LIN {X 0,Y 573.624,Z 371.5,A -85,B 0,C 180,E1 -2266.777,E2 -2266.777} C_VEL
LIN {X 0,Y 573.867,Z 351.071,A -85,B 0,C 180,E1 -2269.438,E2 -2269.438} C_VEL
LIN {X 0,Y 574.138,Z 330.864,A -85,B 0,C 180,E1 -2272.111,E2 -2272.111} C_VEL
LIN {X 0,Y 574.251,Z 318.107,A -85,B 0,C 180,E1 -2273.82,E2 -2273.82} C_VEL
LIN {X 0,Y 573.282,Z 312.704,A -85,B 0,C 180,E1 -2274.609,E2 -2274.609} C_VEL
LIN {X 0,Y 573.246,Z 312.705,A -85,B 0,C 180,E1 -2276.975,E2 -2276.975} C_VEL
LIN {X 0,Y 573.246,Z 312.7,A -85,B 0,C 180,E1 -2279.488,E2 -2279.488} C_VEL
LIN {X 0,Y 573.251,Z 312.707,A -85,B 0,C 180,E1 -2282.644,E2 -2282.644} C_VEL
LIN {X 0,Y 573.249,Z 312.699,A -85,B 0,C 180,E1 -2285.184,E2 -2285.184} C_VEL
LIN {X 0,Y 573.231,Z 312.7,A -85,B 0,C 180,E1 -2287.807,E2 -2287.807} C_VEL
LIN {X 0,Y 573.238,Z 312.706,A -85,B 0,C 180,E1 -2290.524,E2 -2290.524} C_VEL
LIN {X 0,Y 573.232,Z 312.699,A -85,B 0,C 180,E1 -2293.358,E2 -2293.358} C_VEL
LIN {X 0,Y 573.236,Z 312.708,A -85,B 0,C 180,E1 -2296.33,E2 -2296.33} C_VEL
LIN {X 0,Y 573.233,Z 312.705,A -85,B 0,C 180,E1 -2298.543,E2 -2298.543} C_VEL
LIN {X 0,Y 573.231,Z 312.701,A -85,B 0,C 180,E1 -2301.298,E2 -2301.298} C_VEL
LIN {X 0,Y 573.229,Z 312.709,A -85,B 0,C 180,E1 -2304.014,E2 -2304.014} C_VEL
LIN {X 0,Y 573.258,Z 312.7,A -85,B 0,C 180,E1 -2306.517,E2 -2306.517} C_VEL
LIN {X 0,Y 573.214,Z 312.701,A -85,B 0,C 180,E1 -2309.118,E2 -2309.118} C_VEL
LIN {X 0,Y 573.213,Z 312.703,A -85,B 0,C 180,E1 -2311.434,E2 -2311.434} C_VEL
LIN {X 0,Y 573.229,Z 312.701,A -85,B 0,C 180,E1 -2314.589,E2 -2314.589} C_VEL
LIN {X 0,Y 573.216,Z 312.709,A -85,B 0,C 180,E1 -2317.661,E2 -2317.661} C_VEL
LIN {X 0,Y 573.252,Z 312.698,A -85,B 0,C 180,E1 -2320.67,E2 -2320.67} C_VEL
LIN {X 0,Y 573.221,Z 312.71,A -85,B 0,C 180,E1 -2323.621,E2 -2323.621} C_VEL
LIN {X 0,Y 573.245,Z 312.706,A -85,B 0,C 180,E1 -2325.806,E2 -2325.806} C_VEL
LIN {X 0,Y 573.21,Z 312.702,A -85,B 0,C 180,E1 -2328.764,E2 -2328.764} C_VEL
LIN {X 0,Y 573.219,Z 312.711,A -85,B 0,C 180,E1 -2331.54,E2 -2331.54} C_VEL
LIN {X 0,Y 573.245,Z 312.699,A -85,B 0,C 180,E1 -2334.372,E2 -2334.372} C_VEL
LIN {X 0,Y 573.283,Z 312.7,A -85,B 0,C 180,E1 -2337.189,E2 -2337.189} C_VEL
LIN {X 0,Y 573.285,Z 312.695,A -85,B 0,C 180,E1 -2340,E2 -2340} C_VEL
LIN {X 0,Y 573.275,Z 312.696,A -85,B 0,C 180,E1 -2342.811,E2 -2342.811} C_VEL
LIN {X 0,Y 573.272,Z 312.699,A -85,B 0,C 180,E1 -2345.629,E2 -2345.629} C_VEL
LIN {X 0,Y 573.252,Z 312.699,A -85,B 0,C 180,E1 -2347.751,E2 -2347.751} C_VEL
LIN {X 0,Y 573.229,Z 312.703,A -85,B 0,C 180,E1 -2350.598,E2 -2350.598} C_VEL
LIN {X 0,Y 573.223,Z 312.704,A -85,B 0,C 180,E1 -2352.75,E2 -2352.75} C_VEL
LIN {X 0,Y 573.216,Z 312.71,A -85,B 0,C 180,E1 -2354.921,E2 -2354.921} C_VEL
LIN {X 0,Y 573.225,Z 312.701,A -85,B 0,C 180,E1 -2357.849,E2 -2357.849} C_VEL
LIN {X 0,Y 573.228,Z 312.7,A -85,B 0,C 180,E1 -2360.078,E2 -2360.078} C_VEL
LIN {X 0,Y 573.223,Z 312.703,A -85,B 0,C 180,E1 -2362.339,E2 -2362.339} C_VEL
LIN {X 0,Y 573.234,Z 312.702,A -85,B 0,C 180,E1 -2364.358,E2 -2364.358} C_VEL
LIN {X 0,Y 572.608,Z 312.787,A -85,B 0,C 180,E1 -2364.944,E2 -2364.944} C_VEL
LIN {X 0,Y 569.771,Z 313.141,A -85,B 0,C 180,E1 -2365.895,E2 -2365.895} C_VEL
LIN {X 0,Y 567.341,Z 313.441,A -85,B 0,C 180,E1 -2366.661,E2 -2366.661} C_VEL
LIN {X 0,Y 566.286,Z 313.569,A -85,B 0,C 180,E1 -2367.252,E2 -2367.252} C_VEL
LIN {X 0,Y 566.195,Z 313.578,A -85,B 0,C 180,E1 -2367.452,E2 -2367.452} C_VEL
LIN {X 0,Y 566.189,Z 313.578,A -85,B 0,C 180,E1 -2369.77,E2 -2369.77} C_VEL
LIN {X 0,Y 566.198,Z 313.581,A -85,B 0,C 180,E1 -2372.431,E2 -2372.431} C_VEL
LIN {X 0,Y 566.179,Z 313.583,A -85,B 0,C 180,E1 -2374.991,E2 -2374.991} C_VEL
LIN {X 0,Y 566.189,Z 313.577,A -85,B 0,C 180,E1 -2377.462,E2 -2377.462} C_VEL
LIN {X 0,Y 566.221,Z 313.578,A -85,B 0,C 180,E1 -2380.198,E2 -2380.198} C_VEL
LIN {X 0,Y 566.201,Z 313.578,A -85,B 0,C 180,E1 -2383.055,E2 -2383.055} C_VEL
LIN {X 0,Y 566.191,Z 313.582,A -85,B 0,C 180,E1 -2386.05,E2 -2386.05} C_VEL
LIN {X 0,Y 566.218,Z 313.575,A -85,B 0,C 180,E1 -2389.214,E2 -2389.214} C_VEL
LIN {X 0,Y 566.187,Z 313.58,A -85,B 0,C 180,E1 -2391.638,E2 -2391.638} C_VEL
LIN {X 0,Y 566.198,Z 313.585,A -85,B 0,C 180,E1 -2394.312,E2 -2394.312} C_VEL
LIN {X 0,Y 566.229,Z 313.575,A -85,B 0,C 180,E1 -2396.899,E2 -2396.899} C_VEL
LIN {X 0,Y 566.182,Z 313.581,A -85,B 0,C 180,E1 -2399.408,E2 -2399.408} C_VEL
LIN {X 0,Y 566.267,Z 313.716,A -85,B 0,C 180,E1 -2402.514,E2 -2402.514} C_VEL
LIN {X 0,Y 566.832,Z 317.946,A -85,B 0,C 180,E1 -2403.217,E2 -2403.217} C_VEL
LIN {X 0,Y 566.597,Z 335.971,A -85,B 0,C 180,E1 -2406.033,E2 -2406.033} C_VEL
LIN {X 0,Y 566.549,Z 342.685,A -85,B 0,C 180,E1 -2407.072,E2 -2407.072} C_VEL
LIN {X 0,Y 567.797,Z 350.391,A -85,B 0,C 180,E1 -2407.22,E2 -2407.22} C_VEL
LIN {X 0,Y 567.418,Z 479.258,A -85,B 0,C 180,E1 -2408.888,E2 -2408.888} C_VEL
LIN {X 0,Y 567.304,Z 493.234,A -85,B 0,C 180,E1 -2409.207,E2 -2409.207} C_VEL
LIN {X 0,Y 567.147,Z 507.772,A -85,B 0,C 180,E1 -2409.698,E2 -2409.698} C_VEL
LIN {X 0,Y 566.966,Z 520.604,A -85,B 0,C 180,E1 -2410.278,E2 -2410.278} C_VEL
LIN {X 0,Y 566.796,Z 533.294,A -85,B 0,C 180,E1 -2411.005,E2 -2411.005} C_VEL
LIN {X 0,Y 566.583,Z 545.097,A -85,B 0,C 180,E1 -2411.842,E2 -2411.842} C_VEL
LIN {X 0,Y 566.392,Z 556.565,A -85,B 0,C 180,E1 -2412.834,E2 -2412.834} C_VEL
LIN {X 0,Y 566.255,Z 565.673,A -85,B 0,C 180,E1 -2413.785,E2 -2413.785} C_VEL
LIN {X 0,Y 566.162,Z 574.547,A -85,B 0,C 180,E1 -2414.89,E2 -2414.89} C_VEL
LIN {X 0,Y 566.053,Z 582.989,A -85,B 0,C 180,E1 -2416.173,E2 -2416.173} C_VEL
LIN {X 0,Y 565.957,Z 589.719,A -85,B 0,C 180,E1 -2417.449,E2 -2417.449} C_VEL
LIN {X 0,Y 565.963,Z 595.363,A -85,B 0,C 180,E1 -2418.817,E2 -2418.817} C_VEL
LIN {X 0,Y 565.925,Z 599.074,A -85,B 0,C 180,E1 -2419.988,E2 -2419.988} C_VEL
LIN {X 0,Y 565.854,Z 602.252,A -85,B 0,C 180,E1 -2421.429,E2 -2421.429} C_VEL
LIN {X 0,Y 565.886,Z 604.025,A -85,B 0,C 180,E1 -2422.866,E2 -2422.866} C_VEL
LIN {X 0,Y 565.898,Z 604.451,A -85,B 0,C 180,E1 -2424.298,E2 -2424.298} C_VEL
LIN {X 0,Y 565.91,Z 603.55,A -85,B 0,C 180,E1 -2425.727,E2 -2425.727} C_VEL
LIN {X 0,Y 565.872,Z 601.307,A -85,B 0,C 180,E1 -2427.152,E2 -2427.152} C_VEL
LIN {X 0,Y 565.869,Z 597.676,A -85,B 0,C 180,E1 -2428.577,E2 -2428.577} C_VEL
LIN {X 0,Y 565.914,Z 592.561,A -85,B 0,C 180,E1 -2430,E2 -2430} C_VEL
LIN {X 0,Y 566.006,Z 587.613,A -85,B 0,C 180,E1 -2431.067,E2 -2431.067} C_VEL
LIN {X 0,Y 566.042,Z 580.556,A -85,B 0,C 180,E1 -2432.313,E2 -2432.313} C_VEL
LIN {X 0,Y 566.184,Z 573.191,A -85,B 0,C 180,E1 -2433.38,E2 -2433.38} C_VEL
LIN {X 0,Y 566.313,Z 564.376,A -85,B 0,C 180,E1 -2434.448,E2 -2434.448} C_VEL
LIN {X 0,Y 566.456,Z 553.745,A -85,B 0,C 180,E1 -2435.518,E2 -2435.518} C_VEL
LIN {X 0,Y 566.63,Z 543.012,A -85,B 0,C 180,E1 -2436.409,E2 -2436.409} C_VEL
LIN {X 0,Y 566.798,Z 530.428,A -85,B 0,C 180,E1 -2437.267,E2 -2437.267} C_VEL
LIN {X 0,Y 567.034,Z 518.388,A -85,B 0,C 180,E1 -2437.925,E2 -2437.925} C_VEL
LIN {X 0,Y 567.209,Z 504.85,A -85,B 0,C 180,E1 -2438.506,E2 -2438.506} C_VEL
LIN {X 0,Y 567.387,Z 490.587,A -85,B 0,C 180,E1 -2438.952,E2 -2438.952} C_VEL
LIN {X 0,Y 567.466,Z 476.634,A -85,B 0,C 180,E1 -2439.242,E2 -2439.242} C_VEL
LIN {X 0,Y 567.739,Z 349.084,A -85,B 0,C 180,E1 -2440.889,E2 -2440.889} C_VEL
LIN {X 0,Y 566.57,Z 342.666,A -85,B 0,C 180,E1 -2441.021,E2 -2441.021} C_VEL
LIN {X 0,Y 566.763,Z 324.714,A -85,B 0,C 180,E1 -2443.81,E2 -2443.81} C_VEL
LIN {X 0,Y 566.778,Z 316.589,A -85,B 0,C 180,E1 -2445.093,E2 -2445.093} C_VEL
LIN {X 0,Y 566.204,Z 313.585,A -85,B 0,C 180,E1 -2445.616,E2 -2445.616} C_VEL
LIN {X 0,Y 566.206,Z 313.585,A -85,B 0,C 180,E1 -2448.077,E2 -2448.077} C_VEL
LIN {X 0,Y 566.21,Z 313.58,A -85,B 0,C 180,E1 -2450.337,E2 -2450.337} C_VEL
LIN {X 0,Y 566.172,Z 313.582,A -85,B 0,C 180,E1 -2453.28,E2 -2453.28} C_VEL
LIN {X 0,Y 566.217,Z 313.584,A -85,B 0,C 180,E1 -2455.748,E2 -2455.748} C_VEL
LIN {X 0,Y 566.204,Z 313.578,A -85,B 0,C 180,E1 -2458.201,E2 -2458.201} C_VEL
LIN {X 0,Y 566.195,Z 313.579,A -85,B 0,C 180,E1 -2461.076,E2 -2461.076} C_VEL
LIN {X 0,Y 566.213,Z 313.583,A -85,B 0,C 180,E1 -2463.733,E2 -2463.733} C_VEL
LIN {X 0,Y 566.207,Z 313.575,A -85,B 0,C 180,E1 -2466.568,E2 -2466.568} C_VEL
LIN {X 0,Y 566.219,Z 313.578,A -85,B 0,C 180,E1 -2469.685,E2 -2469.685} C_VEL
LIN {X 0,Y 566.197,Z 313.578,A -85,B 0,C 180,E1 -2472.916,E2 -2472.916} C_VEL
LIN {X 0,Y 566.194,Z 313.578,A -85,B 0,C 180,E1 -2476.048,E2 -2476.048} C_VEL
LIN {X 0,Y 566.198,Z 313.583,A -85,B 0,C 180,E1 -2479.213,E2 -2479.213} C_VEL
LIN {X 0,Y 566.178,Z 313.582,A -85,B 0,C 180,E1 -2481.636,E2 -2481.636} C_VEL
LIN {X 0,Y 566.157,Z 313.582,A -85,B 0,C 180,E1 -2484.307,E2 -2484.307} C_VEL
LIN {X 0,Y 566.195,Z 313.581,A -85,B 0,C 180,E1 -2486.896,E2 -2486.896} C_VEL
LIN {X 0,Y 566.169,Z 313.586,A -85,B 0,C 180,E1 -2489.406,E2 -2489.406} C_VEL
LIN {X 0,Y 566.202,Z 313.574,A -85,B 0,C 180,E1 -2491.856,E2 -2491.856} C_VEL
LIN {X 0,Y 566.194,Z 313.576,A -85,B 0,C 180,E1 -2494.25,E2 -2494.25} C_VEL
LIN {X 0,Y 566.161,Z 313.584,A -85,B 0,C 180,E1 -2497.367,E2 -2497.367} C_VEL
LIN {X 0,Y 566.191,Z 313.575,A -85,B 0,C 180,E1 -2499.662,E2 -2499.662} C_VEL
LIN {X 0,Y 566.179,Z 313.584,A -85,B 0,C 180,E1 -2502.667,E2 -2502.667} C_VEL
LIN {X 0,Y 566.2,Z 313.575,A -85,B 0,C 180,E1 -2505.626,E2 -2505.626} C_VEL
LIN {X 0,Y 566.219,Z 313.579,A -85,B 0,C 180,E1 -2508.676,E2 -2508.676} C_VEL
LIN {X 0,Y 566.177,Z 313.58,A -85,B 0,C 180,E1 -2511.433,E2 -2511.433} C_VEL
LIN {X 0,Y 566.233,Z 313.575,A -85,B 0,C 180,E1 -2514.301,E2 -2514.301} C_VEL
LIN {X 0,Y 566.245,Z 313.57,A -85,B 0,C 180,E1 -2517.866,E2 -2517.866} C_VEL
LIN {X 0,Y 566.285,Z 313.572,A -85,B 0,C 180,E1 -2520.711,E2 -2520.711} C_VEL
LIN {X 0,Y 566.242,Z 313.574,A -85,B 0,C 180,E1 -2522.845,E2 -2522.845} C_VEL
LIN {X 0,Y 566.214,Z 313.575,A -85,B 0,C 180,E1 -2525.699,E2 -2525.699} C_VEL
LIN {X 0,Y 566.175,Z 313.584,A -85,B 0,C 180,E1 -2528.566,E2 -2528.566} C_VEL
LIN {X 0,Y 566.224,Z 313.573,A -85,B 0,C 180,E1 -2531.454,E2 -2531.454} C_VEL
LIN {X 0,Y 566.213,Z 313.579,A -85,B 0,C 180,E1 -2534.504,E2 -2534.504} C_VEL
LIN {X 0,Y 566.177,Z 313.579,A -85,B 0,C 180,E1 -2537.332,E2 -2537.332} C_VEL
LIN {X 0,Y 566.191,Z 313.582,A -85,B 0,C 180,E1 -2540.338,E2 -2540.338} C_VEL
LIN {X 0,Y 566.154,Z 313.582,A -85,B 0,C 180,E1 -2543.281,E2 -2543.281} C_VEL
LIN {X 0,Y 566.192,Z 313.581,A -85,B 0,C 180,E1 -2545.75,E2 -2545.75} C_VEL
LIN {X 0,Y 566.171,Z 313.579,A -85,B 0,C 180,E1 -2548.954,E2 -2548.954} C_VEL
LIN {X 0,Y 566.181,Z 313.58,A -85,B 0,C 180,E1 -2551.422,E2 -2551.422} C_VEL
LIN {X 0,Y 566.198,Z 313.585,A -85,B 0,C 180,E1 -2553.957,E2 -2553.957} C_VEL
LIN {X 0,Y 566.198,Z 313.577,A -85,B 0,C 180,E1 -2556.57,E2 -2556.57} C_VEL
LIN {X 0,Y 566.206,Z 313.584,A -85,B 0,C 180,E1 -2559.687,E2 -2559.687} C_VEL
LIN {X 0,Y 566.204,Z 313.58,A -85,B 0,C 180,E1 -2562.088,E2 -2562.088} C_VEL
LIN {X 0,Y 566.166,Z 313.582,A -85,B 0,C 180,E1 -2565.037,E2 -2565.037} C_VEL
LIN {X 0,Y 566.205,Z 313.578,A -85,B 0,C 180,E1 -2568.137,E2 -2568.137} C_VEL
LIN {X 0,Y 566.209,Z 313.576,A -85,B 0,C 180,E1 -2570.727,E2 -2570.727} C_VEL
LIN {X 0,Y 566.202,Z 313.583,A -85,B 0,C 180,E1 -2573.786,E2 -2573.786} C_VEL
LIN {X 0,Y 566.225,Z 313.576,A -85,B 0,C 180,E1 -2576.899,E2 -2576.899} C_VEL
LIN {X 0,Y 566.178,Z 313.589,A -85,B 0,C 180,E1 -2579.408,E2 -2579.408} C_VEL
LIN {X 0,Y 566.209,Z 313.579,A -85,B 0,C 180,E1 -2581.858,E2 -2581.858} C_VEL
LIN {X 0,Y 566.212,Z 313.578,A -85,B 0,C 180,E1 -2584.252,E2 -2584.252} C_VEL
LIN {X 0,Y 566.254,Z 313.637,A -85,B 0,C 180,E1 -2585.237,E2 -2585.237} C_VEL
LIN {X 0,Y 567.336,Z 319.335,A -85,B 0,C 180,E1 -2586.06,E2 -2586.06} C_VEL
LIN {X 0,Y 567.182,Z 336.23,A -85,B 0,C 180,E1 -2588.331,E2 -2588.331} C_VEL
LIN {X 0,Y 566.868,Z 357.712,A -85,B 0,C 180,E1 -2591.196,E2 -2591.196} C_VEL
LIN {X 0,Y 566.675,Z 371.558,A -85,B 0,C 180,E1 -2593.018,E2 -2593.018} C_VEL
LIN {X 0,Y 567.771,Z 378.47,A -85,B 0,C 180,E1 -2593.149,E2 -2593.149} C_VEL
LIN {X 0,Y 567.456,Z 509.907,A -85,B 0,C 180,E1 -2594.856,E2 -2594.856} C_VEL
LIN {X 0,Y 567.276,Z 524.486,A -85,B 0,C 180,E1 -2595.199,E2 -2595.199} C_VEL
LIN {X 0,Y 567.123,Z 538.848,A -85,B 0,C 180,E1 -2595.696,E2 -2595.696} C_VEL
LIN {X 0,Y 566.966,Z 551.65,A -85,B 0,C 180,E1 -2596.287,E2 -2596.287} C_VEL
LIN {X 0,Y 566.772,Z 564.108,A -85,B 0,C 180,E1 -2597.012,E2 -2597.012} C_VEL
LIN {X 0,Y 566.573,Z 576.648,A -85,B 0,C 180,E1 -2597.918,E2 -2597.918} C_VEL
LIN {X 0,Y 566.445,Z 587.322,A -85,B 0,C 180,E1 -2598.861,E2 -2598.861} C_VEL
LIN {X 0,Y 566.206,Z 597.854,A -85,B 0,C 180,E1 -2599.993,E2 -2599.993} C_VEL
LIN {X 0,Y 566.132,Z 606.175,A -85,B 0,C 180,E1 -2601.073,E2 -2601.073} C_VEL
LIN {X 0,Y 566.046,Z 614.129,A -85,B 0,C 180,E1 -2602.33,E2 -2602.33} C_VEL
LIN {X 0,Y 565.943,Z 620.529,A -85,B 0,C 180,E1 -2603.583,E2 -2603.583} C_VEL
LIN {X 0,Y 565.928,Z 624.961,A -85,B 0,C 180,E1 -2604.656,E2 -2604.656} C_VEL
LIN {X 0,Y 565.956,Z 628.444,A -85,B 0,C 180,E1 -2605.727,E2 -2605.727} C_VEL
LIN {X 0,Y 565.874,Z 631.832,A -85,B 0,C 180,E1 -2607.153,E2 -2607.153} C_VEL
LIN {X 0,Y 565.84,Z 633.833,A -85,B 0,C 180,E1 -2608.577,E2 -2608.577} C_VEL
LIN {X 0,Y 565.837,Z 634.5,A -85,B 0,C 180,E1 -2610,E2 -2610} C_VEL
LIN {X 0,Y 565.84,Z 633.834,A -85,B 0,C 180,E1 -2611.423,E2 -2611.423} C_VEL
LIN {X 0,Y 565.874,Z 631.834,A -85,B 0,C 180,E1 -2612.847,E2 -2612.847} C_VEL
LIN {X 0,Y 565.956,Z 628.446,A -85,B 0,C 180,E1 -2614.273,E2 -2614.273} C_VEL
LIN {X 0,Y 565.988,Z 623.569,A -85,B 0,C 180,E1 -2615.701,E2 -2615.701} C_VEL
LIN {X 0,Y 565.992,Z 619.045,A -85,B 0,C 180,E1 -2616.739,E2 -2616.739} C_VEL
LIN {X 0,Y 566.047,Z 612.038,A -85,B 0,C 180,E1 -2618.029,E2 -2618.029} C_VEL
LIN {X 0,Y 566.177,Z 603.56,A -85,B 0,C 180,E1 -2619.286,E2 -2619.286} C_VEL
LIN {X 0,Y 566.294,Z 594.71,A -85,B 0,C 180,E1 -2620.367,E2 -2620.367} C_VEL
LIN {X 0,Y 566.484,Z 583.992,A -85,B 0,C 180,E1 -2621.449,E2 -2621.449} C_VEL
LIN {X 0,Y 566.607,Z 573.144,A -85,B 0,C 180,E1 -2622.354,E2 -2622.354} C_VEL
LIN {X 0,Y 566.779,Z 561.261,A -85,B 0,C 180,E1 -2623.17,E2 -2623.17} C_VEL
LIN {X 0,Y 567.023,Z 548.103,A -85,B 0,C 180,E1 -2623.895,E2 -2623.895} C_VEL
LIN {X 0,Y 567.216,Z 535.036,A -85,B 0,C 180,E1 -2624.454,E2 -2624.454} C_VEL
LIN {X 0,Y 567.354,Z 521.137,A -85,B 0,C 180,E1 -2624.894,E2 -2624.894} C_VEL
LIN {X 0,Y 567.459,Z 507.157,A -85,B 0,C 180,E1 -2625.19,E2 -2625.19} C_VEL
LIN {X 0,Y 567.691,Z 377.288,A -85,B 0,C 180,E1 -2626.869,E2 -2626.869} C_VEL
LIN {X 0,Y 566.675,Z 371.558,A -85,B 0,C 180,E1 -2626.982,E2 -2626.982} C_VEL
LIN {X 0,Y 566.965,Z 350.789,A -85,B 0,C 180,E1 -2629.722,E2 -2629.722} C_VEL
LIN {X 0,Y 567.252,Z 329.377,A -85,B 0,C 180,E1 -2632.586,E2 -2632.586} C_VEL
LIN {X 0,Y 567.335,Z 319.207,A -85,B 0,C 180,E1 -2633.957,E2 -2633.957} C_VEL
LIN {X 0,Y 566.238,Z 313.582,A -85,B 0,C 180,E1 -2634.789,E2 -2634.789} C_VEL
LIN {X 0,Y 566.206,Z 313.578,A -85,B 0,C 180,E1 -2637.339,E2 -2637.339} C_VEL
LIN {X 0,Y 566.199,Z 313.578,A -85,B 0,C 180,E1 -2639.768,E2 -2639.768} C_VEL
LIN {X 0,Y 566.202,Z 313.585,A -85,B 0,C 180,E1 -2642.429,E2 -2642.429} C_VEL
LIN {X 0,Y 566.197,Z 313.579,A -85,B 0,C 180,E1 -2644.992,E2 -2644.992} C_VEL
LIN {X 0,Y 566.191,Z 313.575,A -85,B 0,C 180,E1 -2647.46,E2 -2647.46} C_VEL
LIN {X 0,Y 566.201,Z 313.582,A -85,B 0,C 180,E1 -2650.198,E2 -2650.198} C_VEL
LIN {X 0,Y 566.194,Z 313.577,A -85,B 0,C 180,E1 -2653.053,E2 -2653.053} C_VEL
LIN {X 0,Y 566.19,Z 313.582,A -85,B 0,C 180,E1 -2656.048,E2 -2656.048} C_VEL
LIN {X 0,Y 566.172,Z 313.581,A -85,B 0,C 180,E1 -2658.86,E2 -2658.86} C_VEL
LIN {X 0,Y 566.176,Z 313.582,A -85,B 0,C 180,E1 -2661.636,E2 -2661.636} C_VEL
LIN {X 0,Y 566.181,Z 313.584,A -85,B 0,C 180,E1 -2664.309,E2 -2664.309} C_VEL
LIN {X 0,Y 566.209,Z 313.575,A -85,B 0,C 180,E1 -2666.897,E2 -2666.897} C_VEL
LIN {X 0,Y 566.166,Z 313.58,A -85,B 0,C 180,E1 -2669.406,E2 -2669.406} C_VEL
LIN {X 0,Y 566.174,Z 313.585,A -85,B 0,C 180,E1 -2671.855,E2 -2671.855} C_VEL
LIN {X 0,Y 566.191,Z 313.581,A -85,B 0,C 180,E1 -2674.25,E2 -2674.25} C_VEL
LIN {X 0,Y 566.154,Z 313.582,A -85,B 0,C 180,E1 -2676.719,E2 -2676.719} C_VEL
LIN {X 0,Y 566.19,Z 313.585,A -85,B 0,C 180,E1 -2679.662,E2 -2679.662} C_VEL
LIN {X 0,Y 566.173,Z 313.579,A -85,B 0,C 180,E1 -2682.668,E2 -2682.668} C_VEL
LIN {X 0,Y 566.21,Z 313.584,A -85,B 0,C 180,E1 -2685.626,E2 -2685.626} C_VEL
LIN {X 0,Y 566.173,Z 313.578,A -85,B 0,C 180,E1 -2688.699,E2 -2688.699} C_VEL
LIN {X 0,Y 566.172,Z 313.588,A -85,B 0,C 180,E1 -2691.434,E2 -2691.434} C_VEL
LIN {X 0,Y 566.215,Z 313.574,A -85,B 0,C 180,E1 -2694.301,E2 -2694.301} C_VEL
LIN {X 0,Y 566.247,Z 313.576,A -85,B 0,C 180,E1 -2697.155,E2 -2697.155} C_VEL
LIN {X 0,Y 566.256,Z 313.571,A -85,B 0,C 180,E1 -2700,E2 -2700} C_VEL
LIN {X 0,Y 566.243,Z 313.572,A -85,B 0,C 180,E1 -2702.846,E2 -2702.846} C_VEL
LIN {X 0,Y 566.237,Z 313.574,A -85,B 0,C 180,E1 -2705.699,E2 -2705.699} C_VEL
LIN {X 0,Y 566.18,Z 313.579,A -85,B 0,C 180,E1 -2708.567,E2 -2708.567} C_VEL
LIN {X 0,Y 566.229,Z 313.576,A -85,B 0,C 180,E1 -2711.455,E2 -2711.455} C_VEL
LIN {X 0,Y 566.204,Z 313.578,A -85,B 0,C 180,E1 -2714.5,E2 -2714.5} C_VEL
LIN {X 0,Y 566.184,Z 313.583,A -85,B 0,C 180,E1 -2717.332,E2 -2717.332} C_VEL
LIN {X 0,Y 566.194,Z 313.578,A -85,B 0,C 180,E1 -2720.338,E2 -2720.338} C_VEL
LIN {X 0,Y 566.16,Z 313.585,A -85,B 0,C 180,E1 -2723.282,E2 -2723.282} C_VEL
LIN {X 0,Y 566.202,Z 313.576,A -85,B 0,C 180,E1 -2725.75,E2 -2725.75} C_VEL
LIN {X 0,Y 566.195,Z 313.578,A -85,B 0,C 180,E1 -2727.452,E2 -2727.452} C_VEL
LIN {X 0,Y 565.512,Z 313.662,A -85,B 0,C 180,E1 -2728.046,E2 -2728.046} C_VEL
LIN {X 0,Y 562.647,Z 314.025,A -85,B 0,C 180,E1 -2729.009,E2 -2729.009} C_VEL
LIN {X 0,Y 560.239,Z 314.322,A -85,B 0,C 180,E1 -2729.785,E2 -2729.785} C_VEL
LIN {X 0,Y 559.212,Z 314.451,A -85,B 0,C 180,E1 -2730.384,E2 -2730.384} C_VEL
LIN {X 0,Y 559.132,Z 314.458,A -85,B 0,C 180,E1 -2730.586,E2 -2730.586} C_VEL
LIN {X 0,Y 559.167,Z 314.462,A -85,B 0,C 180,E1 -2732.715,E2 -2732.715} C_VEL
LIN {X 0,Y 559.123,Z 314.459,A -85,B 0,C 180,E1 -2735.325,E2 -2735.325} C_VEL
LIN {X 0,Y 559.128,Z 314.458,A -85,B 0,C 180,E1 -2738.019,E2 -2738.019} C_VEL
LIN {X 0,Y 559.168,Z 314.458,A -85,B 0,C 180,E1 -2740.812,E2 -2740.812} C_VEL
LIN {X 0,Y 559.14,Z 314.457,A -85,B 0,C 180,E1 -2743.735,E2 -2743.735} C_VEL
LIN {X 0,Y 559.141,Z 314.46,A -85,B 0,C 180,E1 -2746.805,E2 -2746.805} C_VEL
LIN {X 0,Y 559.171,Z 314.453,A -85,B 0,C 180,E1 -2749.19,E2 -2749.19} C_VEL
LIN {X 0,Y 559.133,Z 314.462,A -85,B 0,C 180,E1 -2751.984,E2 -2751.984} C_VEL
LIN {X 0,Y 559.153,Z 314.456,A -85,B 0,C 180,E1 -2754.785,E2 -2754.785} C_VEL
LIN {X 0,Y 559.173,Z 314.454,A -85,B 0,C 180,E1 -2757.363,E2 -2757.363} C_VEL
LIN {X 0,Y 559.15,Z 314.464,A -85,B 0,C 180,E1 -2760.143,E2 -2760.143} C_VEL
LIN {X 0,Y 559.237,Z 314.561,A -85,B 0,C 180,E1 -2762.343,E2 -2762.343} C_VEL
LIN {X 0,Y 559.898,Z 319.268,A -85,B 0,C 180,E1 -2763.136,E2 -2763.136} C_VEL
LIN {X 0,Y 559.633,Z 336.681,A -85,B 0,C 180,E1 -2765.913,E2 -2765.913} C_VEL
LIN {X 0,Y 559.599,Z 342.691,A -85,B 0,C 180,E1 -2766.855,E2 -2766.855} C_VEL
LIN {X 0,Y 561,Z 351.323,A -85,B 0,C 180,E1 -2767.022,E2 -2767.022} C_VEL
LIN {X 0,Y 560.577,Z 479.602,A -85,B 0,C 180,E1 -2768.705,E2 -2768.705} C_VEL
LIN {X 0,Y 560.45,Z 493.743,A -85,B 0,C 180,E1 -2769.037,E2 -2769.037} C_VEL
LIN {X 0,Y 560.309,Z 506.99,A -85,B 0,C 180,E1 -2769.487,E2 -2769.487} C_VEL
LIN {X 0,Y 560.097,Z 518.71,A -85,B 0,C 180,E1 -2770.006,E2 -2770.006} C_VEL
LIN {X 0,Y 559.88,Z 531.15,A -85,B 0,C 180,E1 -2770.703,E2 -2770.703} C_VEL
LIN {X 0,Y 559.684,Z 542.881,A -85,B 0,C 180,E1 -2771.515,E2 -2771.515} C_VEL
LIN {X 0,Y 559.446,Z 554.022,A -85,B 0,C 180,E1 -2772.453,E2 -2772.453} C_VEL
LIN {X 0,Y 559.251,Z 564.972,A -85,B 0,C 180,E1 -2773.576,E2 -2773.576} C_VEL
LIN {X 0,Y 559.101,Z 573.961,A -85,B 0,C 180,E1 -2774.694,E2 -2774.694} C_VEL
LIN {X 0,Y 559.01,Z 581.494,A -85,B 0,C 180,E1 -2775.826,E2 -2775.826} C_VEL
LIN {X 0,Y 558.908,Z 587.54,A -85,B 0,C 180,E1 -2776.919,E2 -2776.919} C_VEL
LIN {X 0,Y 558.85,Z 592.599,A -85,B 0,C 180,E1 -2778.024,E2 -2778.024} C_VEL
LIN {X 0,Y 558.832,Z 597.786,A -85,B 0,C 180,E1 -2779.493,E2 -2779.493} C_VEL
LIN {X 0,Y 558.755,Z 600.682,A -85,B 0,C 180,E1 -2780.589,E2 -2780.589} C_VEL
LIN {X 0,Y 558.797,Z 603.224,A -85,B 0,C 180,E1 -2782.048,E2 -2782.048} C_VEL
LIN {X 0,Y 558.848,Z 604.387,A -85,B 0,C 180,E1 -2783.501,E2 -2783.501} C_VEL
LIN {X 0,Y 558.76,Z 604.216,A -85,B 0,C 180,E1 -2784.949,E2 -2784.949} C_VEL
LIN {X 0,Y 558.819,Z 602.715,A -85,B 0,C 180,E1 -2786.395,E2 -2786.395} C_VEL
LIN {X 0,Y 558.748,Z 599.857,A -85,B 0,C 180,E1 -2787.838,E2 -2787.838} C_VEL
LIN {X 0,Y 558.792,Z 595.572,A -85,B 0,C 180,E1 -2789.279,E2 -2789.279} C_VEL
LIN {X 0,Y 558.845,Z 589.741,A -85,B 0,C 180,E1 -2790.721,E2 -2790.721} C_VEL
LIN {X 0,Y 558.961,Z 583.192,A -85,B 0,C 180,E1 -2791.981,E2 -2791.981} C_VEL
LIN {X 0,Y 559.106,Z 575.093,A -85,B 0,C 180,E1 -2793.243,E2 -2793.243} C_VEL
LIN {X 0,Y 559.19,Z 566.66,A -85,B 0,C 180,E1 -2794.325,E2 -2794.325} C_VEL
LIN {X 0,Y 559.41,Z 556.476,A -85,B 0,C 180,E1 -2795.407,E2 -2795.407} C_VEL
LIN {X 0,Y 559.653,Z 545.137,A -85,B 0,C 180,E1 -2796.399,E2 -2796.399} C_VEL
LIN {X 0,Y 559.825,Z 532.59,A -85,B 0,C 180,E1 -2797.295,E2 -2797.295} C_VEL
LIN {X 0,Y 560.098,Z 519.849,A -85,B 0,C 180,E1 -2798.024,E2 -2798.024} C_VEL
LIN {X 0,Y 560.324,Z 506.785,A -85,B 0,C 180,E1 -2798.611,E2 -2798.611} C_VEL
LIN {X 0,Y 560.491,Z 492.652,A -85,B 0,C 180,E1 -2799.086,E2 -2799.086} C_VEL
LIN {X 0,Y 560.623,Z 478.619,A -85,B 0,C 180,E1 -2799.402,E2 -2799.402} C_VEL
LIN {X 0,Y 560.897,Z 349.744,A -85,B 0,C 180,E1 -2801.092,E2 -2801.092} C_VEL
LIN {X 0,Y 559.579,Z 342.603,A -85,B 0,C 180,E1 -2801.249,E2 -2801.249} C_VEL
LIN {X 0,Y 559.833,Z 325.308,A -85,B 0,C 180,E1 -2803.984,E2 -2803.984} C_VEL
LIN {X 0,Y 559.716,Z 317.271,A -85,B 0,C 180,E1 -2805.288,E2 -2805.288} C_VEL
LIN {X 0,Y 559.171,Z 314.461,A -85,B 0,C 180,E1 -2805.771,E2 -2805.771} C_VEL
LIN {X 0,Y 559.151,Z 314.461,A -85,B 0,C 180,E1 -2808.314,E2 -2808.314} C_VEL
LIN {X 0,Y 559.179,Z 314.454,A -85,B 0,C 180,E1 -2810.604,E2 -2810.604} C_VEL
LIN {X 0,Y 559.138,Z 314.464,A -85,B 0,C 180,E1 -2813.716,E2 -2813.716} C_VEL
LIN {X 0,Y 559.183,Z 314.456,A -85,B 0,C 180,E1 -2816.096,E2 -2816.096} C_VEL
LIN {X 0,Y 559.164,Z 314.453,A -85,B 0,C 180,E1 -2818.529,E2 -2818.529} C_VEL
LIN {X 0,Y 559.15,Z 314.458,A -85,B 0,C 180,E1 -2821.273,E2 -2821.273} C_VEL
LIN {X 0,Y 559.168,Z 314.457,A -85,B 0,C 180,E1 -2823.948,E2 -2823.948} C_VEL
LIN {X 0,Y 559.158,Z 314.453,A -85,B 0,C 180,E1 -2826.446,E2 -2826.446} C_VEL
LIN {X 0,Y 559.176,Z 314.453,A -85,B 0,C 180,E1 -2828.933,E2 -2828.933} C_VEL
LIN {X 0,Y 559.16,Z 314.458,A -85,B 0,C 180,E1 -2831.769,E2 -2831.769} C_VEL
LIN {X 0,Y 559.134,Z 314.457,A -85,B 0,C 180,E1 -2834.738,E2 -2834.738} C_VEL
LIN {X 0,Y 559.153,Z 314.462,A -85,B 0,C 180,E1 -2837.255,E2 -2837.255} C_VEL
LIN {X 0,Y 559.173,Z 314.452,A -85,B 0,C 180,E1 -2840.133,E2 -2840.133} C_VEL
LIN {X 0,Y 559.133,Z 314.459,A -85,B 0,C 180,E1 -2842.89,E2 -2842.89} C_VEL
LIN {X 0,Y 559.149,Z 314.454,A -85,B 0,C 180,E1 -2846.051,E2 -2846.051} C_VEL
LIN {X 0,Y 559.147,Z 314.461,A -85,B 0,C 180,E1 -2848.98,E2 -2848.98} C_VEL
LIN {X 0,Y 559.135,Z 314.456,A -85,B 0,C 180,E1 -2851.622,E2 -2851.622} C_VEL
LIN {X 0,Y 559.165,Z 314.452,A -85,B 0,C 180,E1 -2853.902,E2 -2853.902} C_VEL
LIN {X 0,Y 559.106,Z 314.468,A -85,B 0,C 180,E1 -2857.066,E2 -2857.066} C_VEL
LIN {X 0,Y 559.161,Z 314.453,A -85,B 0,C 180,E1 -2859.394,E2 -2859.394} C_VEL
LIN {X 0,Y 559.122,Z 314.458,A -85,B 0,C 180,E1 -2861.685,E2 -2861.685} C_VEL
LIN {X 0,Y 559.141,Z 314.455,A -85,B 0,C 180,E1 -2863.947,E2 -2863.947} C_VEL
LIN {X 0,Y 559.144,Z 314.455,A -85,B 0,C 180,E1 -2866.183,E2 -2866.183} C_VEL
LIN {X 0,Y 559.19,Z 314.453,A -85,B 0,C 180,E1 -2868.605,E2 -2868.605} C_VEL
LIN {X 0,Y 559.173,Z 314.453,A -85,B 0,C 180,E1 -2872.053,E2 -2872.053} C_VEL
LIN {X 0,Y 559.223,Z 314.446,A -85,B 0,C 180,E1 -2874.953,E2 -2874.953} C_VEL
LIN {X 0,Y 559.218,Z 314.446,A -85,B 0,C 180,E1 -2877.839,E2 -2877.839} C_VEL
LIN {X 0,Y 559.255,Z 314.447,A -85,B 0,C 180,E1 -2880.72,E2 -2880.72} C_VEL
LIN {X 0,Y 559.207,Z 314.449,A -85,B 0,C 180,E1 -2882.881,E2 -2882.881} C_VEL
LIN {X 0,Y 559.185,Z 314.451,A -85,B 0,C 180,E1 -2885.77,E2 -2885.77} C_VEL
LIN {X 0,Y 559.141,Z 314.458,A -85,B 0,C 180,E1 -2888.675,E2 -2888.675} C_VEL
LIN {X 0,Y 559.186,Z 314.45,A -85,B 0,C 180,E1 -2891.601,E2 -2891.601} C_VEL
LIN {X 0,Y 559.186,Z 314.453,A -85,B 0,C 180,E1 -2894.596,E2 -2894.596} C_VEL
LIN {X 0,Y 559.121,Z 314.459,A -85,B 0,C 180,E1 -2897.558,E2 -2897.558} C_VEL
LIN {X 0,Y 559.151,Z 314.459,A -85,B 0,C 180,E1 -2899.838,E2 -2899.838} C_VEL
LIN {X 0,Y 559.125,Z 314.466,A -85,B 0,C 180,E1 -2902.153,E2 -2902.153} C_VEL
LIN {X 0,Y 559.161,Z 314.453,A -85,B 0,C 180,E1 -2905.299,E2 -2905.299} C_VEL
LIN {X 0,Y 559.114,Z 314.463,A -85,B 0,C 180,E1 -2907.716,E2 -2907.716} C_VEL
LIN {X 0,Y 559.14,Z 314.461,A -85,B 0,C 180,E1 -2910.183,E2 -2910.183} C_VEL
LIN {X 0,Y 559.146,Z 314.455,A -85,B 0,C 180,E1 -2912.716,E2 -2912.716} C_VEL
LIN {X 0,Y 559.132,Z 314.458,A -85,B 0,C 180,E1 -2915.324,E2 -2915.324} C_VEL
LIN {X 0,Y 559.123,Z 314.465,A -85,B 0,C 180,E1 -2918.018,E2 -2918.018} C_VEL
LIN {X 0,Y 559.15,Z 314.453,A -85,B 0,C 180,E1 -2920.813,E2 -2920.813} C_VEL
LIN {X 0,Y 559.151,Z 314.464,A -85,B 0,C 180,E1 -2923.733,E2 -2923.733} C_VEL
LIN {X 0,Y 559.139,Z 314.456,A -85,B 0,C 180,E1 -2926.804,E2 -2926.804} C_VEL
LIN {X 0,Y 559.151,Z 314.458,A -85,B 0,C 180,E1 -2929.189,E2 -2929.189} C_VEL
LIN {X 0,Y 559.128,Z 314.462,A -85,B 0,C 180,E1 -2931.983,E2 -2931.983} C_VEL
LIN {X 0,Y 559.141,Z 314.457,A -85,B 0,C 180,E1 -2934.678,E2 -2934.678} C_VEL
LIN {X 0,Y 559.17,Z 314.461,A -85,B 0,C 180,E1 -2937.362,E2 -2937.362} C_VEL
LIN {X 0,Y 559.146,Z 314.457,A -85,B 0,C 180,E1 -2940.143,E2 -2940.143} C_VEL
LIN {X 0,Y 559.167,Z 314.46,A -85,B 0,C 180,E1 -2943.098,E2 -2943.098} C_VEL
LIN {X 0,Y 559.221,Z 314.526,A -85,B 0,C 180,E1 -2945.052,E2 -2945.052} C_VEL
LIN {X 0,Y 560.436,Z 320.645,A -85,B 0,C 180,E1 -2945.95,E2 -2945.95} C_VEL
LIN {X 0,Y 560.272,Z 336.382,A -85,B 0,C 180,E1 -2948.091,E2 -2948.091} C_VEL
LIN {X 0,Y 559.947,Z 357.712,A -85,B 0,C 180,E1 -2950.954,E2 -2950.954} C_VEL
LIN {X 0,Y 559.729,Z 371.549,A -85,B 0,C 180,E1 -2952.8,E2 -2952.8} C_VEL
LIN {X 0,Y 560.994,Z 379.126,A -85,B 0,C 180,E1 -2952.948,E2 -2952.948} C_VEL
LIN {X 0,Y 560.622,Z 508.662,A -85,B 0,C 180,E1 -2954.644,E2 -2954.644} C_VEL
LIN {X 0,Y 560.473,Z 522.728,A -85,B 0,C 180,E1 -2954.961,E2 -2954.961} C_VEL
LIN {X 0,Y 560.299,Z 536.493,A -85,B 0,C 180,E1 -2955.421,E2 -2955.421} C_VEL
LIN {X 0,Y 560.087,Z 549.883,A -85,B 0,C 180,E1 -2956.022,E2 -2956.022} C_VEL
LIN {X 0,Y 559.842,Z 562.682,A -85,B 0,C 180,E1 -2956.756,E2 -2956.756} C_VEL
LIN {X 0,Y 559.642,Z 574.315,A -85,B 0,C 180,E1 -2957.582,E2 -2957.582} C_VEL
LIN {X 0,Y 559.43,Z 584.921,A -85,B 0,C 180,E1 -2958.492,E2 -2958.492} C_VEL
LIN {X 0,Y 559.272,Z 594.709,A -85,B 0,C 180,E1 -2959.502,E2 -2959.502} C_VEL
LIN {X 0,Y 559.121,Z 603.56,A -85,B 0,C 180,E1 -2960.596,E2 -2960.596} C_VEL
LIN {X 0,Y 558.985,Z 612.037,A -85,B 0,C 180,E1 -2961.869,E2 -2961.869} C_VEL
LIN {X 0,Y 558.901,Z 618.867,A -85,B 0,C 180,E1 -2963.14,E2 -2963.14} C_VEL
LIN {X 0,Y 558.912,Z 623.57,A -85,B 0,C 180,E1 -2964.227,E2 -2964.227} C_VEL
LIN {X 0,Y 558.865,Z 628.444,A -85,B 0,C 180,E1 -2965.673,E2 -2965.673} C_VEL
LIN {X 0,Y 558.796,Z 631.832,A -85,B 0,C 180,E1 -2967.116,E2 -2967.116} C_VEL
LIN {X 0,Y 558.74,Z 633.834,A -85,B 0,C 180,E1 -2968.559,E2 -2968.559} C_VEL
LIN {X 0,Y 558.738,Z 634.5,A -85,B 0,C 180,E1 -2970,E2 -2970} C_VEL
LIN {X 0,Y 558.74,Z 633.834,A -85,B 0,C 180,E1 -2971.441,E2 -2971.441} C_VEL
LIN {X 0,Y 558.796,Z 631.835,A -85,B 0,C 180,E1 -2972.884,E2 -2972.884} C_VEL
LIN {X 0,Y 558.865,Z 628.446,A -85,B 0,C 180,E1 -2974.327,E2 -2974.327} C_VEL
LIN {X 0,Y 558.917,Z 623.568,A -85,B 0,C 180,E1 -2975.773,E2 -2975.773} C_VEL
LIN {X 0,Y 558.906,Z 617.055,A -85,B 0,C 180,E1 -2977.224,E2 -2977.224} C_VEL
LIN {X 0,Y 559.028,Z 609.803,A -85,B 0,C 180,E1 -2978.495,E2 -2978.495} C_VEL
LIN {X 0,Y 559.146,Z 600.824,A -85,B 0,C 180,E1 -2979.769,E2 -2979.769} C_VEL
LIN {X 0,Y 559.35,Z 591.395,A -85,B 0,C 180,E1 -2980.863,E2 -2980.863} C_VEL
LIN {X 0,Y 559.517,Z 580.957,A -85,B 0,C 180,E1 -2981.869,E2 -2981.869} C_VEL
LIN {X 0,Y 559.709,Z 569.437,A -85,B 0,C 180,E1 -2982.786,E2 -2982.786} C_VEL
LIN {X 0,Y 559.963,Z 556.647,A -85,B 0,C 180,E1 -2983.611,E2 -2983.611} C_VEL
LIN {X 0,Y 560.163,Z 544.157,A -85,B 0,C 180,E1 -2984.254,E2 -2984.254} C_VEL
LIN {X 0,Y 560.408,Z 531.086,A -85,B 0,C 180,E1 -2984.774,E2 -2984.774} C_VEL
LIN {X 0,Y 560.506,Z 517.552,A -85,B 0,C 180,E1 -2985.171,E2 -2985.171} C_VEL
LIN {X 0,Y 560.627,Z 502.632,A -85,B 0,C 180,E1 -2985.449,E2 -2985.449} C_VEL
LIN {X 0,Y 560.919,Z 378.265,A -85,B 0,C 180,E1 -2987.066,E2 -2987.066} C_VEL
LIN {X 0,Y 559.721,Z 371.605,A -85,B 0,C 180,E1 -2987.193,E2 -2987.193} C_VEL
LIN {X 0,Y 560.049,Z 350.627,A -85,B 0,C 180,E1 -2989.996,E2 -2989.996} C_VEL
LIN {X 0,Y 560.438,Z 327.786,A -85,B 0,C 180,E1 -2993.071,E2 -2993.071} C_VEL
LIN {X 0,Y 560.435,Z 320.64,A -85,B 0,C 180,E1 -2994.05,E2 -2994.05} C_VEL
LIN {X 0,Y 559.197,Z 314.459,A -85,B 0,C 180,E1 -2994.975,E2 -2994.975} C_VEL
LIN {X 0,Y 559.153,Z 314.456,A -85,B 0,C 180,E1 -2997.713,E2 -2997.713} C_VEL
LIN {X 0,Y 559.151,Z 314.46,A -85,B 0,C 180,E1 -3000.182,E2 -3000.182} C_VEL
LIN {X 0,Y 559.154,Z 314.462,A -85,B 0,C 180,E1 -3002.714,E2 -3002.714} C_VEL
LIN {X 0,Y 559.141,Z 314.456,A -85,B 0,C 180,E1 -3005.322,E2 -3005.322} C_VEL
LIN {X 0,Y 559.128,Z 314.459,A -85,B 0,C 180,E1 -3008.017,E2 -3008.017} C_VEL
LIN {X 0,Y 559.151,Z 314.456,A -85,B 0,C 180,E1 -3010.811,E2 -3010.811} C_VEL
LIN {X 0,Y 559.139,Z 314.455,A -85,B 0,C 180,E1 -3013.196,E2 -3013.196} C_VEL
LIN {X 0,Y 559.151,Z 314.464,A -85,B 0,C 180,E1 -3016.267,E2 -3016.267} C_VEL
LIN {X 0,Y 559.15,Z 314.454,A -85,B 0,C 180,E1 -3019.187,E2 -3019.187} C_VEL
LIN {X 0,Y 559.123,Z 314.465,A -85,B 0,C 180,E1 -3021.982,E2 -3021.982} C_VEL
LIN {X 0,Y 559.134,Z 314.457,A -85,B 0,C 180,E1 -3024.785,E2 -3024.785} C_VEL
LIN {X 0,Y 559.145,Z 314.456,A -85,B 0,C 180,E1 -3027.364,E2 -3027.364} C_VEL
LIN {X 0,Y 559.135,Z 314.46,A -85,B 0,C 180,E1 -3030.142,E2 -3030.142} C_VEL
LIN {X 0,Y 559.131,Z 314.457,A -85,B 0,C 180,E1 -3033.178,E2 -3033.178} C_VEL
LIN {X 0,Y 559.142,Z 314.459,A -85,B 0,C 180,E1 -3035.494,E2 -3035.494} C_VEL
LIN {X 0,Y 559.157,Z 314.453,A -85,B 0,C 180,E1 -3038.623,E2 -3038.623} C_VEL
LIN {X 0,Y 559.145,Z 314.455,A -85,B 0,C 180,E1 -3040.926,E2 -3040.926} C_VEL
LIN {X 0,Y 559.138,Z 314.461,A -85,B 0,C 180,E1 -3043.947,E2 -3043.947} C_VEL
LIN {X 0,Y 559.141,Z 314.458,A -85,B 0,C 180,E1 -3046.183,E2 -3046.183} C_VEL
LIN {X 0,Y 559.142,Z 314.457,A -85,B 0,C 180,E1 -3049.133,E2 -3049.133} C_VEL
LIN {X 0,Y 559.12,Z 314.459,A -85,B 0,C 180,E1 -3052.053,E2 -3052.053} C_VEL
LIN {X 0,Y 559.229,Z 314.447,A -85,B 0,C 180,E1 -3054.953,E2 -3054.953} C_VEL
LIN {X 0,Y 559.222,Z 314.448,A -85,B 0,C 180,E1 -3057.84,E2 -3057.84} C_VEL
LIN {X 0,Y 559.226,Z 314.447,A -85,B 0,C 180,E1 -3060,E2 -3060} C_VEL
LIN {X 0,Y 559.212,Z 314.449,A -85,B 0,C 180,E1 -3062.882,E2 -3062.882} C_VEL
LIN {X 0,Y 559.204,Z 314.45,A -85,B 0,C 180,E1 -3065.771,E2 -3065.771} C_VEL
LIN {X 0,Y 559.146,Z 314.456,A -85,B 0,C 180,E1 -3068.675,E2 -3068.675} C_VEL
LIN {X 0,Y 559.191,Z 314.45,A -85,B 0,C 180,E1 -3071.601,E2 -3071.601} C_VEL
LIN {X 0,Y 559.168,Z 314.455,A -85,B 0,C 180,E1 -3074.588,E2 -3074.588} C_VEL
LIN {X 0,Y 559.127,Z 314.459,A -85,B 0,C 180,E1 -3077.558,E2 -3077.558} C_VEL
LIN {X 0,Y 559.153,Z 314.454,A -85,B 0,C 180,E1 -3079.838,E2 -3079.838} C_VEL
LIN {X 0,Y 559.129,Z 314.458,A -85,B 0,C 180,E1 -3082.154,E2 -3082.154} C_VEL
LIN {X 0,Y 559.165,Z 314.456,A -85,B 0,C 180,E1 -3085.299,E2 -3085.299} C_VEL
LIN {X 0,Y 559.147,Z 314.454,A -85,B 0,C 180,E1 -3087.714,E2 -3087.714} C_VEL
LIN {X 0,Y 559.132,Z 314.458,A -85,B 0,C 180,E1 -3090.586,E2 -3090.586} C_VEL
LIN {X 0,Y 558.472,Z 314.543,A -85,B 0,C 180,E1 -3091.188,E2 -3091.188} C_VEL
LIN {X 0,Y 555.614,Z 314.897,A -85,B 0,C 180,E1 -3092.164,E2 -3092.164} C_VEL
LIN {X 0,Y 553.203,Z 315.201,A -85,B 0,C 180,E1 -3092.95,E2 -3092.95} C_VEL
LIN {X 0,Y 552.181,Z 315.323,A -85,B 0,C 180,E1 -3093.557,E2 -3093.557} C_VEL
LIN {X 0,Y 552.105,Z 315.332,A -85,B 0,C 180,E1 -3093.762,E2 -3093.762} C_VEL
LIN {X 0,Y 552.098,Z 315.34,A -85,B 0,C 180,E1 -3096.748,E2 -3096.748} C_VEL
LIN {X 0,Y 552.128,Z 315.329,A -85,B 0,C 180,E1 -3099.528,E2 -3099.528} C_VEL
LIN {X 0,Y 552.125,Z 315.338,A -85,B 0,C 180,E1 -3102.427,E2 -3102.427} C_VEL
LIN {X 0,Y 552.092,Z 315.335,A -85,B 0,C 180,E1 -3105.564,E2 -3105.564} C_VEL
LIN {X 0,Y 552.129,Z 315.335,A -85,B 0,C 180,E1 -3108.678,E2 -3108.678} C_VEL
LIN {X 0,Y 552.118,Z 315.331,A -85,B 0,C 180,E1 -3111.412,E2 -3111.412} C_VEL
LIN {X 0,Y 552.103,Z 315.341,A -85,B 0,C 180,E1 -3114.159,E2 -3114.159} C_VEL
LIN {X 0,Y 552.123,Z 315.333,A -85,B 0,C 180,E1 -3116.816,E2 -3116.816} C_VEL
LIN {X 0,Y 552.104,Z 315.335,A -85,B 0,C 180,E1 -3119.392,E2 -3119.392} C_VEL
LIN {X 0,Y 552.17,Z 315.403,A -85,B 0,C 180,E1 -3122.164,E2 -3122.164} C_VEL
LIN {X 0,Y 552.975,Z 321.372,A -85,B 0,C 180,E1 -3123.182,E2 -3123.182} C_VEL
LIN {X 0,Y 552.661,Z 338.73,A -85,B 0,C 180,E1 -3125.988,E2 -3125.988} C_VEL
LIN {X 0,Y 552.629,Z 342.74,A -85,B 0,C 180,E1 -3126.631,E2 -3126.631} C_VEL
LIN {X 0,Y 554.228,Z 352.259,A -85,B 0,C 180,E1 -3126.82,E2 -3126.82} C_VEL
LIN {X 0,Y 553.755,Z 479.173,A -85,B 0,C 180,E1 -3128.503,E2 -3128.503} C_VEL
LIN {X 0,Y 553.596,Z 493.463,A -85,B 0,C 180,E1 -3128.838,E2 -3128.838} C_VEL
LIN {X 0,Y 553.433,Z 507.363,A -85,B 0,C 180,E1 -3129.318,E2 -3129.318} C_VEL
LIN {X 0,Y 553.144,Z 520.811,A -85,B 0,C 180,E1 -3129.938,E2 -3129.938} C_VEL
LIN {X 0,Y 552.888,Z 533.75,A -85,B 0,C 180,E1 -3130.702,E2 -3130.702} C_VEL
LIN {X 0,Y 552.634,Z 545.471,A -85,B 0,C 180,E1 -3131.559,E2 -3131.559} C_VEL
LIN {X 0,Y 552.427,Z 555.788,A -85,B 0,C 180,E1 -3132.472,E2 -3132.472} C_VEL
LIN {X 0,Y 552.22,Z 565.936,A -85,B 0,C 180,E1 -3133.551,E2 -3133.551} C_VEL
LIN {X 0,Y 552.041,Z 574.76,A -85,B 0,C 180,E1 -3134.683,E2 -3134.683} C_VEL
LIN {X 0,Y 551.887,Z 583.15,A -85,B 0,C 180,E1 -3135.998,E2 -3135.998} C_VEL
LIN {X 0,Y 551.824,Z 588.993,A -85,B 0,C 180,E1 -3137.122,E2 -3137.122} C_VEL
LIN {X 0,Y 551.758,Z 593.741,A -85,B 0,C 180,E1 -3138.241,E2 -3138.241} C_VEL
LIN {X 0,Y 551.724,Z 598.637,A -85,B 0,C 180,E1 -3139.727,E2 -3139.727} C_VEL
LIN {X 0,Y 551.675,Z 601.997,A -85,B 0,C 180,E1 -3141.207,E2 -3141.207} C_VEL
LIN {X 0,Y 551.693,Z 603.922,A -85,B 0,C 180,E1 -3142.681,E2 -3142.681} C_VEL
LIN {X 0,Y 551.712,Z 604.484,A -85,B 0,C 180,E1 -3144.151,E2 -3144.151} C_VEL
LIN {X 0,Y 551.696,Z 603.715,A -85,B 0,C 180,E1 -3145.617,E2 -3145.617} C_VEL
LIN {X 0,Y 551.718,Z 601.609,A -85,B 0,C 180,E1 -3147.079,E2 -3147.079} C_VEL
LIN {X 0,Y 551.67,Z 598.121,A -85,B 0,C 180,E1 -3148.54,E2 -3148.54} C_VEL
LIN {X 0,Y 551.728,Z 593.157,A -85,B 0,C 180,E1 -3150,E2 -3150} C_VEL
LIN {X 0,Y 551.789,Z 586.576,A -85,B 0,C 180,E1 -3151.46,E2 -3151.46} C_VEL
LIN {X 0,Y 551.98,Z 579.268,A -85,B 0,C 180,E1 -3152.737,E2 -3152.737} C_VEL
LIN {X 0,Y 552.17,Z 570.221,A -85,B 0,C 180,E1 -3154.014,E2 -3154.014} C_VEL
LIN {X 0,Y 552.316,Z 560.802,A -85,B 0,C 180,E1 -3155.11,E2 -3155.11} C_VEL
LIN {X 0,Y 552.593,Z 549.342,A -85,B 0,C 180,E1 -3156.206,E2 -3156.206} C_VEL
LIN {X 0,Y 552.807,Z 537.743,A -85,B 0,C 180,E1 -3157.115,E2 -3157.115} C_VEL
LIN {X 0,Y 553.068,Z 526.572,A -85,B 0,C 180,E1 -3157.833,E2 -3157.833} C_VEL
LIN {X 0,Y 553.317,Z 513.906,A -85,B 0,C 180,E1 -3158.491,E2 -3158.491} C_VEL
LIN {X 0,Y 553.521,Z 500.201,A -85,B 0,C 180,E1 -3159.04,E2 -3159.04} C_VEL
LIN {X 0,Y 553.742,Z 485.797,A -85,B 0,C 180,E1 -3159.451,E2 -3159.451} C_VEL
LIN {X 0,Y 553.789,Z 471.624,A -85,B 0,C 180,E1 -3159.703,E2 -3159.703} C_VEL
LIN {X 0,Y 554.19,Z 351.12,A -85,B 0,C 180,E1 -3161.287,E2 -3161.287} C_VEL
LIN {X 0,Y 552.597,Z 342.766,A -85,B 0,C 180,E1 -3161.458,E2 -3161.458} C_VEL
LIN {X 0,Y 552.904,Z 325.991,A -85,B 0,C 180,E1 -3164.163,E2 -3164.163} C_VEL
LIN {X 0,Y 552.929,Z 319.867,A -85,B 0,C 180,E1 -3165.16,E2 -3165.16} C_VEL
LIN {X 0,Y 552.131,Z 315.339,A -85,B 0,C 180,E1 -3165.977,E2 -3165.977} C_VEL
LIN {X 0,Y 552.129,Z 315.333,A -85,B 0,C 180,E1 -3168.555,E2 -3168.555} C_VEL
LIN {X 0,Y 552.121,Z 315.332,A -85,B 0,C 180,E1 -3170.88,E2 -3170.88} C_VEL
LIN {X 0,Y 552.104,Z 315.339,A -85,B 0,C 180,E1 -3174.037,E2 -3174.037} C_VEL
LIN {X 0,Y 552.122,Z 315.332,A -85,B 0,C 180,E1 -3176.456,E2 -3176.456} C_VEL
LIN {X 0,Y 552.11,Z 315.331,A -85,B 0,C 180,E1 -3178.927,E2 -3178.927} C_VEL
LIN {X 0,Y 552.112,Z 315.338,A -85,B 0,C 180,E1 -3181.475,E2 -3181.475} C_VEL
LIN {X 0,Y 552.138,Z 315.33,A -85,B 0,C 180,E1 -3184.17,E2 -3184.17} C_VEL
LIN {X 0,Y 552.108,Z 315.332,A -85,B 0,C 180,E1 -3186.746,E2 -3186.746} C_VEL
LIN {X 0,Y 552.131,Z 315.335,A -85,B 0,C 180,E1 -3189.526,E2 -3189.526} C_VEL
LIN {X 0,Y 552.126,Z 315.329,A -85,B 0,C 180,E1 -3192.424,E2 -3192.424} C_VEL
LIN {X 0,Y 552.093,Z 315.341,A -85,B 0,C 180,E1 -3195.562,E2 -3195.562} C_VEL
LIN {X 0,Y 552.115,Z 315.33,A -85,B 0,C 180,E1 -3198.553,E2 -3198.553} C_VEL
LIN {X 0,Y 552.11,Z 315.338,A -85,B 0,C 180,E1 -3201.41,E2 -3201.41} C_VEL
LIN {X 0,Y 552.079,Z 315.336,A -85,B 0,C 180,E1 -3204.155,E2 -3204.155} C_VEL
LIN {X 0,Y 552.099,Z 315.336,A -85,B 0,C 180,E1 -3206.813,E2 -3206.813} C_VEL
LIN {X 0,Y 552.093,Z 315.339,A -85,B 0,C 180,E1 -3209.39,E2 -3209.39} C_VEL
LIN {X 0,Y 552.086,Z 315.332,A -85,B 0,C 180,E1 -3211.9,E2 -3211.9} C_VEL
LIN {X 0,Y 552.096,Z 315.336,A -85,B 0,C 180,E1 -3214.659,E2 -3214.659} C_VEL
LIN {X 0,Y 552.076,Z 315.336,A -85,B 0,C 180,E1 -3217.548,E2 -3217.548} C_VEL
LIN {X 0,Y 552.132,Z 315.327,A -85,B 0,C 180,E1 -3220.374,E2 -3220.374} C_VEL
LIN {X 0,Y 552.11,Z 315.34,A -85,B 0,C 180,E1 -3222.975,E2 -3222.975} C_VEL
LIN {X 0,Y 552.107,Z 315.33,A -85,B 0,C 180,E1 -3226.003,E2 -3226.003} C_VEL
LIN {X 0,Y 552.138,Z 315.333,A -85,B 0,C 180,E1 -3228.993,E2 -3228.993} C_VEL
LIN {X 0,Y 552.128,Z 315.33,A -85,B 0,C 180,E1 -3231.951,E2 -3231.951} C_VEL
LIN {X 0,Y 552.199,Z 315.322,A -85,B 0,C 180,E1 -3234.888,E2 -3234.888} C_VEL
LIN {X 0,Y 552.191,Z 315.321,A -85,B 0,C 180,E1 -3237.812,E2 -3237.812} C_VEL
LIN {X 0,Y 552.225,Z 315.323,A -85,B 0,C 180,E1 -3240.729,E2 -3240.729} C_VEL
LIN {X 0,Y 552.172,Z 315.325,A -85,B 0,C 180,E1 -3242.918,E2 -3242.918} C_VEL
LIN {X 0,Y 552.157,Z 315.327,A -85,B 0,C 180,E1 -3245.844,E2 -3245.844} C_VEL
LIN {X 0,Y 552.114,Z 315.332,A -85,B 0,C 180,E1 -3248.786,E2 -3248.786} C_VEL
LIN {X 0,Y 552.142,Z 315.329,A -85,B 0,C 180,E1 -3251.751,E2 -3251.751} C_VEL
LIN {X 0,Y 552.121,Z 315.331,A -85,B 0,C 180,E1 -3254.749,E2 -3254.749} C_VEL
LIN {X 0,Y 552.079,Z 315.338,A -85,B 0,C 180,E1 -3257.789,E2 -3257.789} C_VEL
LIN {X 0,Y 552.112,Z 315.34,A -85,B 0,C 180,E1 -3260.102,E2 -3260.102} C_VEL
LIN {X 0,Y 552.077,Z 315.34,A -85,B 0,C 180,E1 -3262.451,E2 -3262.451} C_VEL
LIN {X 0,Y 552.124,Z 315.33,A -85,B 0,C 180,E1 -3265.347,E2 -3265.347} C_VEL
LIN {X 0,Y 552.065,Z 315.345,A -85,B 0,C 180,E1 -3268.101,E2 -3268.101} C_VEL
LIN {X 0,Y 552.089,Z 315.334,A -85,B 0,C 180,E1 -3270.61,E2 -3270.61} C_VEL
LIN {X 0,Y 552.104,Z 315.333,A -85,B 0,C 180,E1 -3273.187,E2 -3273.187} C_VEL
LIN {X 0,Y 552.09,Z 315.343,A -85,B 0,C 180,E1 -3275.843,E2 -3275.843} C_VEL
LIN {X 0,Y 552.112,Z 315.332,A -85,B 0,C 180,E1 -3279.062,E2 -3279.062} C_VEL
LIN {X 0,Y 552.123,Z 315.333,A -85,B 0,C 180,E1 -3281.446,E2 -3281.446} C_VEL
LIN {X 0,Y 552.087,Z 315.334,A -85,B 0,C 180,E1 -3284.533,E2 -3284.533} C_VEL
LIN {X 0,Y 552.124,Z 315.339,A -85,B 0,C 180,E1 -3287.585,E2 -3287.585} C_VEL
LIN {X 0,Y 552.124,Z 315.331,A -85,B 0,C 180,E1 -3290.474,E2 -3290.474} C_VEL
LIN {X 0,Y 552.115,Z 315.339,A -85,B 0,C 180,E1 -3293.316,E2 -3293.316} C_VEL
LIN {X 0,Y 552.125,Z 315.334,A -85,B 0,C 180,E1 -3295.94,E2 -3295.94} C_VEL
LIN {X 0,Y 552.116,Z 315.332,A -85,B 0,C 180,E1 -3298.541,E2 -3298.541} C_VEL
LIN {X 0,Y 552.122,Z 315.338,A -85,B 0,C 180,E1 -3301.439,E2 -3301.439} C_VEL
LIN {X 0,Y 552.129,Z 315.333,A -85,B 0,C 180,E1 -3304.356,E2 -3304.356} C_VEL
LIN {X 0,Y 552.16,Z 315.398,A -85,B 0,C 180,E1 -3304.857,E2 -3304.857} C_VEL
LIN {X 0,Y 553.621,Z 323.309,A -85,B 0,C 180,E1 -3306.033,E2 -3306.033} C_VEL
LIN {X 0,Y 553.235,Z 343.325,A -85,B 0,C 180,E1 -3308.775,E2 -3308.775} C_VEL
LIN {X 0,Y 552.9,Z 364.728,A -85,B 0,C 180,E1 -3311.664,E2 -3311.664} C_VEL
LIN {X 0,Y 552.787,Z 371.556,A -85,B 0,C 180,E1 -3312.578,E2 -3312.578} C_VEL
LIN {X 0,Y 554.225,Z 380.061,A -85,B 0,C 180,E1 -3312.745,E2 -3312.745} C_VEL
LIN {X 0,Y 553.779,Z 509.907,A -85,B 0,C 180,E1 -3314.473,E2 -3314.473} C_VEL
LIN {X 0,Y 553.594,Z 523.836,A -85,B 0,C 180,E1 -3314.804,E2 -3314.804} C_VEL
LIN {X 0,Y 553.378,Z 537.716,A -85,B 0,C 180,E1 -3315.286,E2 -3315.286} C_VEL
LIN {X 0,Y 553.161,Z 551.646,A -85,B 0,C 180,E1 -3315.938,E2 -3315.938} C_VEL
LIN {X 0,Y 552.879,Z 564.106,A -85,B 0,C 180,E1 -3316.68,E2 -3316.68} C_VEL
LIN {X 0,Y 552.624,Z 576.652,A -85,B 0,C 180,E1 -3317.608,E2 -3317.608} C_VEL
LIN {X 0,Y 552.446,Z 587.297,A -85,B 0,C 180,E1 -3318.573,E2 -3318.573} C_VEL
LIN {X 0,Y 552.179,Z 597.855,A -85,B 0,C 180,E1 -3319.736,E2 -3319.736} C_VEL
LIN {X 0,Y 552.032,Z 606.176,A -85,B 0,C 180,E1 -3320.843,E2 -3320.843} C_VEL
LIN {X 0,Y 551.912,Z 614.128,A -85,B 0,C 180,E1 -3322.132,E2 -3322.132} C_VEL
LIN {X 0,Y 551.821,Z 620.529,A -85,B 0,C 180,E1 -3323.418,E2 -3323.418} C_VEL
LIN {X 0,Y 551.792,Z 624.961,A -85,B 0,C 180,E1 -3324.519,E2 -3324.519} C_VEL
LIN {X 0,Y 551.759,Z 628.444,A -85,B 0,C 180,E1 -3325.617,E2 -3325.617} C_VEL
LIN {X 0,Y 551.72,Z 631.832,A -85,B 0,C 180,E1 -3327.079,E2 -3327.079} C_VEL
LIN {X 0,Y 551.64,Z 633.834,A -85,B 0,C 180,E1 -3328.54,E2 -3328.54} C_VEL
LIN {X 0,Y 551.639,Z 634.5,A -85,B 0,C 180,E1 -3330,E2 -3330} C_VEL
LIN {X 0,Y 551.64,Z 633.835,A -85,B 0,C 180,E1 -3331.46,E2 -3331.46} C_VEL
LIN {X 0,Y 551.72,Z 631.835,A -85,B 0,C 180,E1 -3332.921,E2 -3332.921} C_VEL
LIN {X 0,Y 551.759,Z 628.447,A -85,B 0,C 180,E1 -3334.383,E2 -3334.383} C_VEL
LIN {X 0,Y 551.825,Z 623.568,A -85,B 0,C 180,E1 -3335.848,E2 -3335.848} C_VEL
LIN {X 0,Y 551.832,Z 617.055,A -85,B 0,C 180,E1 -3337.317,E2 -3337.317} C_VEL
LIN {X 0,Y 551.962,Z 609.804,A -85,B 0,C 180,E1 -3338.604,E2 -3338.604} C_VEL
LIN {X 0,Y 552.116,Z 600.824,A -85,B 0,C 180,E1 -3339.895,E2 -3339.895} C_VEL
LIN {X 0,Y 552.346,Z 591.395,A -85,B 0,C 180,E1 -3341.003,E2 -3341.003} C_VEL
LIN {X 0,Y 552.538,Z 580.957,A -85,B 0,C 180,E1 -3342.021,E2 -3342.021} C_VEL
LIN {X 0,Y 552.76,Z 569.435,A -85,B 0,C 180,E1 -3342.949,E2 -3342.949} C_VEL
LIN {X 0,Y 553.025,Z 556.646,A -85,B 0,C 180,E1 -3343.785,E2 -3343.785} C_VEL
LIN {X 0,Y 553.284,Z 544.154,A -85,B 0,C 180,E1 -3344.435,E2 -3344.435} C_VEL
LIN {X 0,Y 553.541,Z 530.961,A -85,B 0,C 180,E1 -3344.966,E2 -3344.966} C_VEL
LIN {X 0,Y 553.671,Z 517.412,A -85,B 0,C 180,E1 -3345.366,E2 -3345.366} C_VEL
LIN {X 0,Y 553.78,Z 502.632,A -85,B 0,C 180,E1 -3345.645,E2 -3345.645} C_VEL
LIN {X 0,Y 554.162,Z 379.149,A -85,B 0,C 180,E1 -3347.269,E2 -3347.269} C_VEL
LIN {X 0,Y 552.777,Z 371.52,A -85,B 0,C 180,E1 -3347.427,E2 -3347.427} C_VEL
LIN {X 0,Y 553.111,Z 350.466,A -85,B 0,C 180,E1 -3350.257,E2 -3350.257} C_VEL
LIN {X 0,Y 553.566,Z 327.667,A -85,B 0,C 180,E1 -3353.367,E2 -3353.367} C_VEL
LIN {X 0,Y 553.516,Z 321.884,A -85,B 0,C 180,E1 -3354.171,E2 -3354.171} C_VEL
LIN {X 0,Y 552.157,Z 315.334,A -85,B 0,C 180,E1 -3355.174,E2 -3355.174} C_VEL
LIN {X 0,Y 552.107,Z 315.336,A -85,B 0,C 180,E1 -3358.098,E2 -3358.098} C_VEL
LIN {X 0,Y 552.1,Z 315.342,A -85,B 0,C 180,E1 -3360.608,E2 -3360.608} C_VEL
LIN {X 0,Y 552.112,Z 315.334,A -85,B 0,C 180,E1 -3363.185,E2 -3363.185} C_VEL
LIN {X 0,Y 552.098,Z 315.335,A -85,B 0,C 180,E1 -3365.842,E2 -3365.842} C_VEL
LIN {X 0,Y 552.116,Z 315.331,A -85,B 0,C 180,E1 -3369.06,E2 -3369.06} C_VEL
LIN {X 0,Y 552.123,Z 315.328,A -85,B 0,C 180,E1 -3371.444,E2 -3371.444} C_VEL
LIN {X 0,Y 552.088,Z 315.338,A -85,B 0,C 180,E1 -3374.531,E2 -3374.531} C_VEL
LIN {X 0,Y 552.123,Z 315.33,A -85,B 0,C 180,E1 -3377.584,E2 -3377.584} C_VEL
LIN {X 0,Y 552.12,Z 315.336,A -85,B 0,C 180,E1 -3380.472,E2 -3380.472} C_VEL
LIN {X 0,Y 552.101,Z 315.333,A -85,B 0,C 180,E1 -3383.316,E2 -3383.316} C_VEL
LIN {X 0,Y 552.116,Z 315.338,A -85,B 0,C 180,E1 -3385.938,E2 -3385.938} C_VEL
LIN {X 0,Y 552.108,Z 315.331,A -85,B 0,C 180,E1 -3388.54,E2 -3388.54} C_VEL
LIN {X 0,Y 552.085,Z 315.333,A -85,B 0,C 180,E1 -3391.443,E2 -3391.443} C_VEL
LIN {X 0,Y 552.124,Z 315.329,A -85,B 0,C 180,E1 -3394.653,E2 -3394.653} C_VEL
LIN {X 0,Y 552.076,Z 315.341,A -85,B 0,C 180,E1 -3397.548,E2 -3397.548} C_VEL
LIN {X 0,Y 552.13,Z 315.33,A -85,B 0,C 180,E1 -3400.375,E2 -3400.375} C_VEL
LIN {X 0,Y 552.107,Z 315.332,A -85,B 0,C 180,E1 -3402.976,E2 -3402.976} C_VEL
LIN {X 0,Y 552.11,Z 315.336,A -85,B 0,C 180,E1 -3406.004,E2 -3406.004} C_VEL
LIN {X 0,Y 552.11,Z 315.331,A -85,B 0,C 180,E1 -3408.993,E2 -3408.993} C_VEL
LIN {X 0,Y 552.09,Z 315.336,A -85,B 0,C 180,E1 -3411.951,E2 -3411.951} C_VEL
LIN {X 0,Y 552.203,Z 315.321,A -85,B 0,C 180,E1 -3414.889,E2 -3414.889} C_VEL
LIN {X 0,Y 552.195,Z 315.323,A -85,B 0,C 180,E1 -3417.812,E2 -3417.812} C_VEL
LIN {X 0,Y 552.196,Z 315.322,A -85,B 0,C 180,E1 -3420,E2 -3420} C_VEL
LIN {X 0,Y 552.18,Z 315.325,A -85,B 0,C 180,E1 -3422.919,E2 -3422.919} C_VEL
LIN {X 0,Y 552.172,Z 315.325,A -85,B 0,C 180,E1 -3425.844,E2 -3425.844} C_VEL
LIN {X 0,Y 552.119,Z 315.333,A -85,B 0,C 180,E1 -3428.787,E2 -3428.787} C_VEL
LIN {X 0,Y 552.148,Z 315.326,A -85,B 0,C 180,E1 -3431.751,E2 -3431.751} C_VEL
LIN {X 0,Y 552.116,Z 315.336,A -85,B 0,C 180,E1 -3434.749,E2 -3434.749} C_VEL
LIN {X 0,Y 552.085,Z 315.335,A -85,B 0,C 180,E1 -3437.79,E2 -3437.79} C_VEL
LIN {X 0,Y 552.114,Z 315.331,A -85,B 0,C 180,E1 -3440.102,E2 -3440.102} C_VEL
LIN {X 0,Y 552.081,Z 315.338,A -85,B 0,C 180,E1 -3442.452,E2 -3442.452} C_VEL
LIN {X 0,Y 552.145,Z 315.33,A -85,B 0,C 180,E1 -3445.351,E2 -3445.351} C_VEL
LIN {X 0,Y 552.1,Z 315.333,A -85,B 0,C 180,E1 -3448.099,E2 -3448.099} C_VEL
LIN {X 0,Y 552.095,Z 315.341,A -85,B 0,C 180,E1 -3450.61,E2 -3450.61} C_VEL
LIN {X 0,Y 552.115,Z 315.333,A -85,B 0,C 180,E1 -3453.186,E2 -3453.186} C_VEL
LIN {X 0,Y 552.105,Z 315.332,A -85,B 0,C 180,E1 -3453.762,E2 -3453.762} C_VEL
LIN {X 0,Y 551.466,Z 315.418,A -85,B 0,C 180,E1 -3454.371,E2 -3454.371} C_VEL
LIN {X 0,Y 548.646,Z 315.771,A -85,B 0,C 180,E1 -3455.359,E2 -3455.359} C_VEL
LIN {X 0,Y 546.229,Z 316.073,A -85,B 0,C 180,E1 -3456.154,E2 -3456.154} C_VEL
LIN {X 0,Y 545.16,Z 316.204,A -85,B 0,C 180,E1 -3456.768,E2 -3456.768} C_VEL
LIN {X 0,Y 545.058,Z 316.213,A -85,B 0,C 180,E1 -3456.976,E2 -3456.976} C_VEL
LIN {X 0,Y 545.068,Z 316.212,A -85,B 0,C 180,E1 -3460.143,E2 -3460.143} C_VEL
LIN {X 0,Y 545.074,Z 316.21,A -85,B 0,C 180,E1 -3463.108,E2 -3463.108} C_VEL
LIN {X 0,Y 545.047,Z 316.214,A -85,B 0,C 180,E1 -3465.871,E2 -3465.871} C_VEL
LIN {X 0,Y 545.089,Z 316.21,A -85,B 0,C 180,E1 -3468.887,E2 -3468.887} C_VEL
LIN {X 0,Y 545.052,Z 316.214,A -85,B 0,C 180,E1 -3471.764,E2 -3471.764} C_VEL
LIN {X 0,Y 545.057,Z 316.215,A -85,B 0,C 180,E1 -3474.534,E2 -3474.534} C_VEL
LIN {X 0,Y 545.081,Z 316.209,A -85,B 0,C 180,E1 -3477.213,E2 -3477.213} C_VEL
LIN {X 0,Y 545.065,Z 316.216,A -85,B 0,C 180,E1 -3479.811,E2 -3479.811} C_VEL
LIN {X 0,Y 545.116,Z 316.277,A -85,B 0,C 180,E1 -3481.981,E2 -3481.981} C_VEL
LIN {X 0,Y 546.017,Z 321.86,A -85,B 0,C 180,E1 -3482.954,E2 -3482.954} C_VEL
LIN {X 0,Y 545.764,Z 337.148,A -85,B 0,C 180,E1 -3485.463,E2 -3485.463} C_VEL
LIN {X 0,Y 545.69,Z 343.26,A -85,B 0,C 180,E1 -3486.416,E2 -3486.416} C_VEL
LIN {X 0,Y 547.426,Z 352.353,A -85,B 0,C 180,E1 -3486.597,E2 -3486.597} C_VEL
LIN {X 0,Y 546.912,Z 480.041,A -85,B 0,C 180,E1 -3488.319,E2 -3488.319} C_VEL
LIN {X 0,Y 546.747,Z 494.038,A -85,B 0,C 180,E1 -3488.659,E2 -3488.659} C_VEL
LIN {X 0,Y 546.556,Z 507.775,A -85,B 0,C 180,E1 -3489.144,E2 -3489.144} C_VEL
LIN {X 0,Y 546.244,Z 521.154,A -85,B 0,C 180,E1 -3489.774,E2 -3489.774} C_VEL
LIN {X 0,Y 545.94,Z 533.977,A -85,B 0,C 180,E1 -3490.544,E2 -3490.544} C_VEL
LIN {X 0,Y 545.658,Z 545.657,A -85,B 0,C 180,E1 -3491.412,E2 -3491.412} C_VEL
LIN {X 0,Y 545.424,Z 555.502,A -85,B 0,C 180,E1 -3492.294,E2 -3492.294} C_VEL
LIN {X 0,Y 545.21,Z 565.233,A -85,B 0,C 180,E1 -3493.333,E2 -3493.333} C_VEL
LIN {X 0,Y 544.999,Z 574.176,A -85,B 0,C 180,E1 -3494.48,E2 -3494.48} C_VEL
LIN {X 0,Y 544.841,Z 582.705,A -85,B 0,C 180,E1 -3495.814,E2 -3495.814} C_VEL
LIN {X 0,Y 544.753,Z 588.605,A -85,B 0,C 180,E1 -3496.952,E2 -3496.952} C_VEL
LIN {X 0,Y 544.688,Z 593.437,A -85,B 0,C 180,E1 -3498.086,E2 -3498.086} C_VEL
LIN {X 0,Y 544.639,Z 598.412,A -85,B 0,C 180,E1 -3499.592,E2 -3499.592} C_VEL
LIN {X 0,Y 544.571,Z 601.846,A -85,B 0,C 180,E1 -3501.091,E2 -3501.091} C_VEL
LIN {X 0,Y 544.606,Z 603.856,A -85,B 0,C 180,E1 -3502.586,E2 -3502.586} C_VEL
LIN {X 0,Y 544.617,Z 604.498,A -85,B 0,C 180,E1 -3504.075,E2 -3504.075} C_VEL
LIN {X 0,Y 544.592,Z 603.797,A -85,B 0,C 180,E1 -3505.559,E2 -3505.559} C_VEL
LIN {X 0,Y 544.644,Z 601.759,A -85,B 0,C 180,E1 -3507.041,E2 -3507.041} C_VEL
LIN {X 0,Y 544.571,Z 598.344,A -85,B 0,C 180,E1 -3508.521,E2 -3508.521} C_VEL
LIN {X 0,Y 544.635,Z 593.455,A -85,B 0,C 180,E1 -3510,E2 -3510} C_VEL
LIN {X 0,Y 544.784,Z 588.746,A -85,B 0,C 180,E1 -3511.109,E2 -3511.109} C_VEL
LIN {X 0,Y 544.836,Z 581.953,A -85,B 0,C 180,E1 -3512.403,E2 -3512.403} C_VEL
LIN {X 0,Y 544.94,Z 573.553,A -85,B 0,C 180,E1 -3513.697,E2 -3513.697} C_VEL
LIN {X 0,Y 545.218,Z 564.804,A -85,B 0,C 180,E1 -3514.806,E2 -3514.806} C_VEL
LIN {X 0,Y 545.461,Z 554.252,A -85,B 0,C 180,E1 -3515.916,E2 -3515.916} C_VEL
LIN {X 0,Y 545.732,Z 544.154,A -85,B 0,C 180,E1 -3516.798,E2 -3516.798} C_VEL
LIN {X 0,Y 545.977,Z 532.035,A -85,B 0,C 180,E1 -3517.674,E2 -3517.674} C_VEL
LIN {X 0,Y 546.292,Z 519.308,A -85,B 0,C 180,E1 -3518.415,E2 -3518.415} C_VEL
LIN {X 0,Y 546.573,Z 506.118,A -85,B 0,C 180,E1 -3519.016,E2 -3519.016} C_VEL
LIN {X 0,Y 546.825,Z 492.472,A -85,B 0,C 180,E1 -3519.478,E2 -3519.478} C_VEL
LIN {X 0,Y 546.972,Z 478.249,A -85,B 0,C 180,E1 -3519.802,E2 -3519.802} C_VEL
LIN {X 0,Y 547.443,Z 352.193,A -85,B 0,C 180,E1 -3521.494,E2 -3521.494} C_VEL
LIN {X 0,Y 545.656,Z 342.965,A -85,B 0,C 180,E1 -3521.683,E2 -3521.683} C_VEL
LIN {X 0,Y 545.991,Z 325.488,A -85,B 0,C 180,E1 -3524.536,E2 -3524.536} C_VEL
LIN {X 0,Y 545.925,Z 320.716,A -85,B 0,C 180,E1 -3525.328,E2 -3525.328} C_VEL
LIN {X 0,Y 545.101,Z 316.214,A -85,B 0,C 180,E1 -3526.141,E2 -3526.141} C_VEL
LIN {X 0,Y 545.082,Z 316.21,A -85,B 0,C 180,E1 -3528.804,E2 -3528.804} C_VEL
LIN {X 0,Y 545.068,Z 316.212,A -85,B 0,C 180,E1 -3531.163,E2 -3531.163} C_VEL
LIN {X 0,Y 545.051,Z 316.214,A -85,B 0,C 180,E1 -3534.368,E2 -3534.368} C_VEL
LIN {X 0,Y 545.095,Z 316.208,A -85,B 0,C 180,E1 -3537.172,E2 -3537.172} C_VEL
LIN {X 0,Y 545.064,Z 316.212,A -85,B 0,C 180,E1 -3539.338,E2 -3539.338} C_VEL
LIN {X 0,Y 545.061,Z 316.216,A -85,B 0,C 180,E1 -3541.913,E2 -3541.913} C_VEL
LIN {X 0,Y 545.08,Z 316.207,A -85,B 0,C 180,E1 -3544.562,E2 -3544.562} C_VEL
LIN {X 0,Y 545.037,Z 316.217,A -85,B 0,C 180,E1 -3547.303,E2 -3547.303} C_VEL
LIN {X 0,Y 545.065,Z 316.206,A -85,B 0,C 180,E1 -3550.141,E2 -3550.141} C_VEL
LIN {X 0,Y 545.075,Z 316.212,A -85,B 0,C 180,E1 -3553.105,E2 -3553.105} C_VEL
LIN {X 0,Y 545.063,Z 316.21,A -85,B 0,C 180,E1 -3556.223,E2 -3556.223} C_VEL
LIN {X 0,Y 545.075,Z 316.209,A -85,B 0,C 180,E1 -3558.884,E2 -3558.884} C_VEL
LIN {X 0,Y 545.073,Z 316.211,A -85,B 0,C 180,E1 -3560.817,E2 -3560.817} C_VEL
LIN {X 0,Y 545.035,Z 316.217,A -85,B 0,C 180,E1 -3563.619,E2 -3563.619} C_VEL
LIN {X 0,Y 545.043,Z 316.211,A -85,B 0,C 180,E1 -3566.326,E2 -3566.326} C_VEL
LIN {X 0,Y 545.057,Z 316.216,A -85,B 0,C 180,E1 -3568.951,E2 -3568.951} C_VEL
LIN {X 0,Y 545.074,Z 316.209,A -85,B 0,C 180,E1 -3571.506,E2 -3571.506} C_VEL
LIN {X 0,Y 545.059,Z 316.209,A -85,B 0,C 180,E1 -3573.998,E2 -3573.998} C_VEL
LIN {X 0,Y 545.022,Z 316.219,A -85,B 0,C 180,E1 -3577.241,E2 -3577.241} C_VEL
LIN {X 0,Y 545.103,Z 316.202,A -85,B 0,C 180,E1 -3580.414,E2 -3580.414} C_VEL
LIN {X 0,Y 545.041,Z 316.213,A -85,B 0,C 180,E1 -3583.52,E2 -3583.52} C_VEL
LIN {X 0,Y 545.07,Z 316.206,A -85,B 0,C 180,E1 -3585.819,E2 -3585.819} C_VEL
LIN {X 0,Y 545.096,Z 316.212,A -85,B 0,C 180,E1 -3588.849,E2 -3588.849} C_VEL
LIN {X 0,Y 545.077,Z 316.208,A -85,B 0,C 180,E1 -3591.846,E2 -3591.846} C_VEL
LIN {X 0,Y 545.175,Z 316.197,A -85,B 0,C 180,E1 -3594.822,E2 -3594.822} C_VEL
LIN {X 0,Y 545.164,Z 316.196,A -85,B 0,C 180,E1 -3597.783,E2 -3597.783} C_VEL
LIN {X 0,Y 545.194,Z 316.198,A -85,B 0,C 180,E1 -3600.738,E2 -3600.738} C_VEL
LIN {X 0,Y 545.137,Z 316.2,A -85,B 0,C 180,E1 -3602.956,E2 -3602.956} C_VEL
LIN {X 0,Y 545.109,Z 316.206,A -85,B 0,C 180,E1 -3605.92,E2 -3605.92} C_VEL
LIN {X 0,Y 545.075,Z 316.207,A -85,B 0,C 180,E1 -3608.901,E2 -3608.901} C_VEL
LIN {X 0,Y 545.086,Z 316.209,A -85,B 0,C 180,E1 -3611.905,E2 -3611.905} C_VEL
LIN {X 0,Y 545.07,Z 316.207,A -85,B 0,C 180,E1 -3614.944,E2 -3614.944} C_VEL
LIN {X 0,Y 545.045,Z 316.217,A -85,B 0,C 180,E1 -3618.027,E2 -3618.027} C_VEL
LIN {X 0,Y 545.078,Z 316.211,A -85,B 0,C 180,E1 -3620.373,E2 -3620.373} C_VEL
LIN {X 0,Y 545.065,Z 316.211,A -85,B 0,C 180,E1 -3623.56,E2 -3623.56} C_VEL
LIN {X 0,Y 545.06,Z 316.217,A -85,B 0,C 180,E1 -3626.001,E2 -3626.001} C_VEL
LIN {X 0,Y 545.056,Z 316.21,A -85,B 0,C 180,E1 -3628.745,E2 -3628.745} C_VEL
LIN {X 0,Y 545.046,Z 316.216,A -85,B 0,C 180,E1 -3631.679,E2 -3631.679} C_VEL
LIN {X 0,Y 545.056,Z 316.211,A -85,B 0,C 180,E1 -3634.565,E2 -3634.565} C_VEL
LIN {X 0,Y 545.028,Z 316.216,A -85,B 0,C 180,E1 -3637.305,E2 -3637.305} C_VEL
LIN {X 0,Y 545.057,Z 316.212,A -85,B 0,C 180,E1 -3640.143,E2 -3640.143} C_VEL
LIN {X 0,Y 545.071,Z 316.209,A -85,B 0,C 180,E1 -3643.107,E2 -3643.107} C_VEL
LIN {X 0,Y 545.043,Z 316.214,A -85,B 0,C 180,E1 -3646.227,E2 -3646.227} C_VEL
LIN {X 0,Y 545.079,Z 316.209,A -85,B 0,C 180,E1 -3648.887,E2 -3648.887} C_VEL
LIN {X 0,Y 545.047,Z 316.219,A -85,B 0,C 180,E1 -3651.764,E2 -3651.764} C_VEL
LIN {X 0,Y 545.049,Z 316.213,A -85,B 0,C 180,E1 -3654.534,E2 -3654.534} C_VEL
LIN {X 0,Y 545.078,Z 316.215,A -85,B 0,C 180,E1 -3657.213,E2 -3657.213} C_VEL
LIN {X 0,Y 545.061,Z 316.214,A -85,B 0,C 180,E1 -3659.811,E2 -3659.811} C_VEL
LIN {X 0,Y 545.078,Z 316.21,A -85,B 0,C 180,E1 -3662.344,E2 -3662.344} C_VEL
LIN {X 0,Y 545.118,Z 316.265,A -85,B 0,C 180,E1 -3664.657,E2 -3664.657} C_VEL
LIN {X 0,Y 546.705,Z 324.374,A -85,B 0,C 180,E1 -3665.884,E2 -3665.884} C_VEL
LIN {X 0,Y 546.351,Z 343.13,A -85,B 0,C 180,E1 -3668.494,E2 -3668.494} C_VEL
LIN {X 0,Y 545.961,Z 364.541,A -85,B 0,C 180,E1 -3671.422,E2 -3671.422} C_VEL
LIN {X 0,Y 545.824,Z 371.443,A -85,B 0,C 180,E1 -3672.357,E2 -3672.357} C_VEL
LIN {X 0,Y 547.454,Z 380.858,A -85,B 0,C 180,E1 -3672.538,E2 -3672.538} C_VEL
LIN {X 0,Y 546.944,Z 508.633,A -85,B 0,C 180,E1 -3674.25,E2 -3674.25} C_VEL
LIN {X 0,Y 546.742,Z 523.403,A -85,B 0,C 180,E1 -3674.596,E2 -3674.596} C_VEL
LIN {X 0,Y 546.516,Z 537.714,A -85,B 0,C 180,E1 -3675.097,E2 -3675.097} C_VEL
LIN {X 0,Y 546.258,Z 551.644,A -85,B 0,C 180,E1 -3675.756,E2 -3675.756} C_VEL
LIN {X 0,Y 545.924,Z 564.103,A -85,B 0,C 180,E1 -3676.507,E2 -3676.507} C_VEL
LIN {X 0,Y 545.665,Z 576.654,A -85,B 0,C 180,E1 -3677.447,E2 -3677.447} C_VEL
LIN {X 0,Y 545.432,Z 587.949,A -85,B 0,C 180,E1 -3678.492,E2 -3678.492} C_VEL
LIN {X 0,Y 545.175,Z 597.855,A -85,B 0,C 180,E1 -3679.603,E2 -3679.603} C_VEL
LIN {X 0,Y 544.999,Z 606.176,A -85,B 0,C 180,E1 -3680.724,E2 -3680.724} C_VEL
LIN {X 0,Y 544.833,Z 614.128,A -85,B 0,C 180,E1 -3682.029,E2 -3682.029} C_VEL
LIN {X 0,Y 544.753,Z 620.877,A -85,B 0,C 180,E1 -3683.413,E2 -3683.413} C_VEL
LIN {X 0,Y 544.646,Z 626.201,A -85,B 0,C 180,E1 -3684.818,E2 -3684.818} C_VEL
LIN {X 0,Y 544.657,Z 630.317,A -85,B 0,C 180,E1 -3686.301,E2 -3686.301} C_VEL
LIN {X 0,Y 544.569,Z 633.002,A -85,B 0,C 180,E1 -3687.781,E2 -3687.781} C_VEL
LIN {X 0,Y 544.539,Z 634.333,A -85,B 0,C 180,E1 -3689.261,E2 -3689.261} C_VEL
LIN {X 0,Y 544.539,Z 634.334,A -85,B 0,C 180,E1 -3690.739,E2 -3690.739} C_VEL
LIN {X 0,Y 544.569,Z 633.005,A -85,B 0,C 180,E1 -3692.219,E2 -3692.219} C_VEL
LIN {X 0,Y 544.657,Z 630.32,A -85,B 0,C 180,E1 -3693.699,E2 -3693.699} C_VEL
LIN {X 0,Y 544.646,Z 626.202,A -85,B 0,C 180,E1 -3695.182,E2 -3695.182} C_VEL
LIN {X 0,Y 544.734,Z 620.949,A -85,B 0,C 180,E1 -3696.57,E2 -3696.57} C_VEL
LIN {X 0,Y 544.833,Z 614.128,A -85,B 0,C 180,E1 -3697.971,E2 -3697.971} C_VEL
LIN {X 0,Y 544.998,Z 606.176,A -85,B 0,C 180,E1 -3699.276,E2 -3699.276} C_VEL
LIN {X 0,Y 545.175,Z 597.854,A -85,B 0,C 180,E1 -3700.397,E2 -3700.397} C_VEL
LIN {X 0,Y 545.363,Z 588.029,A -85,B 0,C 180,E1 -3701.501,E2 -3701.501} C_VEL
LIN {X 0,Y 545.661,Z 576.652,A -85,B 0,C 180,E1 -3702.553,E2 -3702.553} C_VEL
LIN {X 0,Y 545.919,Z 564.106,A -85,B 0,C 180,E1 -3703.493,E2 -3703.493} C_VEL
LIN {X 0,Y 546.257,Z 551.645,A -85,B 0,C 180,E1 -3704.244,E2 -3704.244} C_VEL
LIN {X 0,Y 546.52,Z 537.703,A -85,B 0,C 180,E1 -3704.903,E2 -3704.903} C_VEL
LIN {X 0,Y 546.718,Z 523.713,A -85,B 0,C 180,E1 -3705.395,E2 -3705.395} C_VEL
LIN {X 0,Y 546.91,Z 509.875,A -85,B 0,C 180,E1 -3705.727,E2 -3705.727} C_VEL
LIN {X 0,Y 547.42,Z 380.202,A -85,B 0,C 180,E1 -3707.472,E2 -3707.472} C_VEL
LIN {X 0,Y 545.818,Z 371.255,A -85,B 0,C 180,E1 -3707.668,E2 -3707.668} C_VEL
LIN {X 0,Y 546.232,Z 350.27,A -85,B 0,C 180,E1 -3710.524,E2 -3710.524} C_VEL
LIN {X 0,Y 546.671,Z 327.681,A -85,B 0,C 180,E1 -3713.648,E2 -3713.648} C_VEL
LIN {X 0,Y 546.58,Z 323.122,A -85,B 0,C 180,E1 -3714.296,E2 -3714.296} C_VEL
LIN {X 0,Y 545.112,Z 316.211,A -85,B 0,C 180,E1 -3715.366,E2 -3715.366} C_VEL
LIN {X 0,Y 545.099,Z 316.212,A -85,B 0,C 180,E1 -3718.492,E2 -3718.492} C_VEL
LIN {X 0,Y 545.063,Z 316.214,A -85,B 0,C 180,E1 -3721.047,E2 -3721.047} C_VEL
LIN {X 0,Y 545.063,Z 316.211,A -85,B 0,C 180,E1 -3723.671,E2 -3723.671} C_VEL
LIN {X 0,Y 545.072,Z 316.208,A -85,B 0,C 180,E1 -3726.926,E2 -3726.926} C_VEL
LIN {X 0,Y 545.06,Z 316.214,A -85,B 0,C 180,E1 -3730.142,E2 -3730.142} C_VEL
LIN {X 0,Y 545.072,Z 316.207,A -85,B 0,C 180,E1 -3733.106,E2 -3733.106} C_VEL
LIN {X 0,Y 545.049,Z 316.219,A -85,B 0,C 180,E1 -3736.225,E2 -3736.225} C_VEL
LIN {X 0,Y 545.078,Z 316.208,A -85,B 0,C 180,E1 -3738.885,E2 -3738.885} C_VEL
LIN {X 0,Y 545.042,Z 316.216,A -85,B 0,C 180,E1 -3741.762,E2 -3741.762} C_VEL
LIN {X 0,Y 545.04,Z 316.215,A -85,B 0,C 180,E1 -3744.532,E2 -3744.532} C_VEL
LIN {X 0,Y 545.058,Z 316.21,A -85,B 0,C 180,E1 -3747.211,E2 -3747.211} C_VEL
LIN {X 0,Y 545.05,Z 316.214,A -85,B 0,C 180,E1 -3749.81,E2 -3749.81} C_VEL
LIN {X 0,Y 545.034,Z 316.216,A -85,B 0,C 180,E1 -3752.341,E2 -3752.341} C_VEL
LIN {X 0,Y 545.092,Z 316.205,A -85,B 0,C 180,E1 -3754.819,E2 -3754.819} C_VEL
LIN {X 0,Y 545.021,Z 316.216,A -85,B 0,C 180,E1 -3757.242,E2 -3757.242} C_VEL
LIN {X 0,Y 545.102,Z 316.206,A -85,B 0,C 180,E1 -3760.414,E2 -3760.414} C_VEL
LIN {X 0,Y 545.039,Z 316.219,A -85,B 0,C 180,E1 -3763.52,E2 -3763.52} C_VEL
LIN {X 0,Y 545.066,Z 316.216,A -85,B 0,C 180,E1 -3765.819,E2 -3765.819} C_VEL
LIN {X 0,Y 545.059,Z 316.209,A -85,B 0,C 180,E1 -3768.848,E2 -3768.848} C_VEL
LIN {X 0,Y 545.048,Z 316.214,A -85,B 0,C 180,E1 -3771.846,E2 -3771.846} C_VEL
LIN {X 0,Y 545.178,Z 316.196,A -85,B 0,C 180,E1 -3774.823,E2 -3774.823} C_VEL
LIN {X 0,Y 545.168,Z 316.199,A -85,B 0,C 180,E1 -3777.784,E2 -3777.784} C_VEL
LIN {X 0,Y 545.166,Z 316.198,A -85,B 0,C 180,E1 -3780,E2 -3780} C_VEL
LIN {X 0,Y 545.148,Z 316.201,A -85,B 0,C 180,E1 -3782.956,E2 -3782.956} C_VEL
LIN {X 0,Y 545.121,Z 316.203,A -85,B 0,C 180,E1 -3785.92,E2 -3785.92} C_VEL
LIN {X 0,Y 545.079,Z 316.206,A -85,B 0,C 180,E1 -3788.154,E2 -3788.154} C_VEL
LIN {X 0,Y 545.12,Z 316.203,A -85,B 0,C 180,E1 -3791.534,E2 -3791.534} C_VEL
LIN {X 0,Y 545.069,Z 316.217,A -85,B 0,C 180,E1 -3794.944,E2 -3794.944} C_VEL
LIN {X 0,Y 545.057,Z 316.21,A -85,B 0,C 180,E1 -3798.027,E2 -3798.027} C_VEL
LIN {X 0,Y 545.08,Z 316.208,A -85,B 0,C 180,E1 -3800.373,E2 -3800.373} C_VEL
LIN {X 0,Y 545.069,Z 316.209,A -85,B 0,C 180,E1 -3803.56,E2 -3803.56} C_VEL
LIN {X 0,Y 545.069,Z 316.209,A -85,B 0,C 180,E1 -3806.002,E2 -3806.002} C_VEL
LIN {X 0,Y 545.079,Z 316.215,A -85,B 0,C 180,E1 -3808.749,E2 -3808.749} C_VEL
LIN {X 0,Y 545.051,Z 316.21,A -85,B 0,C 180,E1 -3811.68,E2 -3811.68} C_VEL
LIN {X 0,Y 545.066,Z 316.217,A -85,B 0,C 180,E1 -3814.565,E2 -3814.565} C_VEL
LIN {X 0,Y 545.058,Z 316.213,A -85,B 0,C 180,E1 -3816.976,E2 -3816.976} C_VEL
LIN {X 0,Y 544.35,Z 316.3,A -85,B 0,C 180,E1 -3817.592,E2 -3817.592} C_VEL
LIN {X 0,Y 541.487,Z 316.664,A -85,B 0,C 180,E1 -3818.593,E2 -3818.593} C_VEL
LIN {X 0,Y 539.102,Z 316.956,A -85,B 0,C 180,E1 -3819.399,E2 -3819.399} C_VEL
LIN {X 0,Y 538.093,Z 317.08,A -85,B 0,C 180,E1 -3820.021,E2 -3820.021} C_VEL
LIN {X 0,Y 538.017,Z 317.088,A -85,B 0,C 180,E1 -3820.232,E2 -3820.232} C_VEL
LIN {X 0,Y 538.021,Z 317.09,A -85,B 0,C 180,E1 -3822.989,E2 -3822.989} C_VEL
LIN {X 0,Y 538.016,Z 317.091,A -85,B 0,C 180,E1 -3825.928,E2 -3825.928} C_VEL
LIN {X 0,Y 538.048,Z 317.085,A -85,B 0,C 180,E1 -3829.226,E2 -3829.226} C_VEL
LIN {X 0,Y 537.992,Z 317.098,A -85,B 0,C 180,E1 -3832.123,E2 -3832.123} C_VEL
LIN {X 0,Y 538.015,Z 317.088,A -85,B 0,C 180,E1 -3834.918,E2 -3834.918} C_VEL
LIN {X 0,Y 538.027,Z 317.09,A -85,B 0,C 180,E1 -3837.619,E2 -3837.619} C_VEL
LIN {X 0,Y 538.019,Z 317.095,A -85,B 0,C 180,E1 -3840.24,E2 -3840.24} C_VEL
LIN {X 0,Y 538.082,Z 317.127,A -85,B 0,C 180,E1 -3841.794,E2 -3841.794} C_VEL
LIN {X 0,Y 539.099,Z 323.144,A -85,B 0,C 180,E1 -3842.854,E2 -3842.854} C_VEL
LIN {X 0,Y 538.83,Z 338.052,A -85,B 0,C 180,E1 -3845.332,E2 -3845.332} C_VEL
LIN {X 0,Y 538.737,Z 343.128,A -85,B 0,C 180,E1 -3846.167,E2 -3846.167} C_VEL
LIN {X 0,Y 540.701,Z 353.878,A -85,B 0,C 180,E1 -3846.391,E2 -3846.391} C_VEL
LIN {X 0,Y 540.094,Z 479.818,A -85,B 0,C 180,E1 -3848.107,E2 -3848.107} C_VEL
LIN {X 0,Y 539.932,Z 493.964,A -85,B 0,C 180,E1 -3848.451,E2 -3848.451} C_VEL
LIN {X 0,Y 539.699,Z 507.183,A -85,B 0,C 180,E1 -3848.917,E2 -3848.917} C_VEL
LIN {X 0,Y 539.401,Z 520.311,A -85,B 0,C 180,E1 -3849.532,E2 -3849.532} C_VEL
LIN {X 0,Y 539.053,Z 532.919,A -85,B 0,C 180,E1 -3850.285,E2 -3850.285} C_VEL
LIN {X 0,Y 538.76,Z 544.775,A -85,B 0,C 180,E1 -3851.165,E2 -3851.165} C_VEL
LIN {X 0,Y 538.479,Z 555.3,A -85,B 0,C 180,E1 -3852.112,E2 -3852.112} C_VEL
LIN {X 0,Y 538.219,Z 564.57,A -85,B 0,C 180,E1 -3853.11,E2 -3853.11} C_VEL
LIN {X 0,Y 537.974,Z 573.592,A -85,B 0,C 180,E1 -3854.272,E2 -3854.272} C_VEL
LIN {X 0,Y 537.812,Z 582.229,A -85,B 0,C 180,E1 -3855.624,E2 -3855.624} C_VEL
LIN {X 0,Y 537.681,Z 588.217,A -85,B 0,C 180,E1 -3856.777,E2 -3856.777} C_VEL
LIN {X 0,Y 537.605,Z 593.133,A -85,B 0,C 180,E1 -3857.927,E2 -3857.927} C_VEL
LIN {X 0,Y 537.564,Z 598.185,A -85,B 0,C 180,E1 -3859.454,E2 -3859.454} C_VEL
LIN {X 0,Y 537.471,Z 601.692,A -85,B 0,C 180,E1 -3860.973,E2 -3860.973} C_VEL
LIN {X 0,Y 537.518,Z 603.775,A -85,B 0,C 180,E1 -3862.487,E2 -3862.487} C_VEL
LIN {X 0,Y 537.529,Z 604.496,A -85,B 0,C 180,E1 -3863.996,E2 -3863.996} C_VEL
LIN {X 0,Y 537.49,Z 603.876,A -85,B 0,C 180,E1 -3865.5,E2 -3865.5} C_VEL
LIN {X 0,Y 537.545,Z 601.91,A -85,B 0,C 180,E1 -3867.002,E2 -3867.002} C_VEL
LIN {X 0,Y 537.474,Z 598.566,A -85,B 0,C 180,E1 -3868.501,E2 -3868.501} C_VEL
LIN {X 0,Y 537.542,Z 593.753,A -85,B 0,C 180,E1 -3870,E2 -3870} C_VEL
LIN {X 0,Y 537.691,Z 589.124,A -85,B 0,C 180,E1 -3871.123,E2 -3871.123} C_VEL
LIN {X 0,Y 537.773,Z 582.418,A -85,B 0,C 180,E1 -3872.434,E2 -3872.434} C_VEL
LIN {X 0,Y 537.892,Z 574.117,A -85,B 0,C 180,E1 -3873.746,E2 -3873.746} C_VEL
LIN {X 0,Y 538.194,Z 565.514,A -85,B 0,C 180,E1 -3874.869,E2 -3874.869} C_VEL
LIN {X 0,Y 538.464,Z 555.144,A -85,B 0,C 180,E1 -3875.993,E2 -3875.993} C_VEL
LIN {X 0,Y 538.782,Z 543.396,A -85,B 0,C 180,E1 -3877.038,E2 -3877.038} C_VEL
LIN {X 0,Y 539.092,Z 531.977,A -85,B 0,C 180,E1 -3877.867,E2 -3877.867} C_VEL
LIN {X 0,Y 539.425,Z 519.22,A -85,B 0,C 180,E1 -3878.617,E2 -3878.617} C_VEL
LIN {X 0,Y 539.747,Z 505.941,A -85,B 0,C 180,E1 -3879.225,E2 -3879.225} C_VEL
LIN {X 0,Y 540.032,Z 492.086,A -85,B 0,C 180,E1 -3879.693,E2 -3879.693} C_VEL
LIN {X 0,Y 540.131,Z 477.489,A -85,B 0,C 180,E1 -3880.022,E2 -3880.022} C_VEL
LIN {X 0,Y 540.658,Z 352.879,A -85,B 0,C 180,E1 -3881.713,E2 -3881.713} C_VEL
LIN {X 0,Y 538.7,Z 343.13,A -85,B 0,C 180,E1 -3881.922,E2 -3881.922} C_VEL
LIN {X 0,Y 539.094,Z 326.16,A -85,B 0,C 180,E1 -3884.727,E2 -3884.727} C_VEL
LIN {X 0,Y 538.938,Z 321.555,A -85,B 0,C 180,E1 -3885.505,E2 -3885.505} C_VEL
LIN {X 0,Y 538.08,Z 317.088,A -85,B 0,C 180,E1 -3886.308,E2 -3886.308} C_VEL
LIN {X 0,Y 538.039,Z 317.088,A -85,B 0,C 180,E1 -3889.059,E2 -3889.059} C_VEL
LIN {X 0,Y 538.019,Z 317.096,A -85,B 0,C 180,E1 -3891.957,E2 -3891.957} C_VEL
LIN {X 0,Y 538.03,Z 317.087,A -85,B 0,C 180,E1 -3894.708,E2 -3894.708} C_VEL
LIN {X 0,Y 538.06,Z 317.086,A -85,B 0,C 180,E1 -3897.351,E2 -3897.351} C_VEL
LIN {X 0,Y 538.027,Z 317.087,A -85,B 0,C 180,E1 -3900.443,E2 -3900.443} C_VEL
LIN {X 0,Y 538.046,Z 317.087,A -85,B 0,C 180,E1 -3903.282,E2 -3903.282} C_VEL
LIN {X 0,Y 538.023,Z 317.089,A -85,B 0,C 180,E1 -3906.001,E2 -3906.001} C_VEL
LIN {X 0,Y 538.013,Z 317.088,A -85,B 0,C 180,E1 -3908.829,E2 -3908.829} C_VEL
LIN {X 0,Y 538.027,Z 317.091,A -85,B 0,C 180,E1 -3911.772,E2 -3911.772} C_VEL
LIN {X 0,Y 538.026,Z 317.087,A -85,B 0,C 180,E1 -3914.858,E2 -3914.858} C_VEL
LIN {X 0,Y 538.014,Z 317.094,A -85,B 0,C 180,E1 -3917.213,E2 -3917.213} C_VEL
LIN {X 0,Y 538.016,Z 317.088,A -85,B 0,C 180,E1 -3920.202,E2 -3920.202} C_VEL
LIN {X 0,Y 538.017,Z 317.092,A -85,B 0,C 180,E1 -3923.066,E2 -3923.066} C_VEL
LIN {X 0,Y 538.007,Z 317.089,A -85,B 0,C 180,E1 -3925.825,E2 -3925.825} C_VEL
LIN {X 0,Y 538,Z 317.09,A -85,B 0,C 180,E1 -3928.498,E2 -3928.498} C_VEL
LIN {X 0,Y 538.01,Z 317.095,A -85,B 0,C 180,E1 -3931.096,E2 -3931.096} C_VEL
LIN {X 0,Y 538.026,Z 317.086,A -85,B 0,C 180,E1 -3933.632,E2 -3933.632} C_VEL
LIN {X 0,Y 537.999,Z 317.098,A -85,B 0,C 180,E1 -3936.927,E2 -3936.927} C_VEL
LIN {X 0,Y 538.068,Z 317.077,A -85,B 0,C 180,E1 -3940.147,E2 -3940.147} C_VEL
LIN {X 0,Y 537.99,Z 317.094,A -85,B 0,C 180,E1 -3943.298,E2 -3943.298} C_VEL
LIN {X 0,Y 538.042,Z 317.082,A -85,B 0,C 180,E1 -3945.63,E2 -3945.63} C_VEL
LIN {X 0,Y 538.057,Z 317.086,A -85,B 0,C 180,E1 -3948.701,E2 -3948.701} C_VEL
LIN {X 0,Y 538.041,Z 317.084,A -85,B 0,C 180,E1 -3951.739,E2 -3951.739} C_VEL
LIN {X 0,Y 538.131,Z 317.075,A -85,B 0,C 180,E1 -3954.754,E2 -3954.754} C_VEL
LIN {X 0,Y 538.138,Z 317.071,A -85,B 0,C 180,E1 -3957.754,E2 -3957.754} C_VEL
LIN {X 0,Y 538.164,Z 317.074,A -85,B 0,C 180,E1 -3960.748,E2 -3960.748} C_VEL
LIN {X 0,Y 538.102,Z 317.076,A -85,B 0,C 180,E1 -3962.994,E2 -3962.994} C_VEL
LIN {X 0,Y 538.066,Z 317.084,A -85,B 0,C 180,E1 -3965.998,E2 -3965.998} C_VEL
LIN {X 0,Y 538.029,Z 317.084,A -85,B 0,C 180,E1 -3969.018,E2 -3969.018} C_VEL
LIN {X 0,Y 538.045,Z 317.088,A -85,B 0,C 180,E1 -3972.063,E2 -3972.063} C_VEL
LIN {X 0,Y 538.029,Z 317.083,A -85,B 0,C 180,E1 -3975.144,E2 -3975.144} C_VEL
LIN {X 0,Y 537.998,Z 317.098,A -85,B 0,C 180,E1 -3978.271,E2 -3978.271} C_VEL
LIN {X 0,Y 538.023,Z 317.086,A -85,B 0,C 180,E1 -3980.652,E2 -3980.652} C_VEL
LIN {X 0,Y 537.989,Z 317.096,A -85,B 0,C 180,E1 -3983.889,E2 -3983.889} C_VEL
LIN {X 0,Y 538.021,Z 317.09,A -85,B 0,C 180,E1 -3986.368,E2 -3986.368} C_VEL
LIN {X 0,Y 538.018,Z 317.087,A -85,B 0,C 180,E1 -3988.934,E2 -3988.934} C_VEL
LIN {X 0,Y 537.999,Z 317.097,A -85,B 0,C 180,E1 -3991.888,E2 -3991.888} C_VEL
LIN {X 0,Y 538.006,Z 317.089,A -85,B 0,C 180,E1 -3994.619,E2 -3994.619} C_VEL
LIN {X 0,Y 537.996,Z 317.091,A -85,B 0,C 180,E1 -3997.171,E2 -3997.171} C_VEL
LIN {X 0,Y 538.014,Z 317.095,A -85,B 0,C 180,E1 -3999.798,E2 -3999.798} C_VEL
LIN {X 0,Y 538.011,Z 317.087,A -85,B 0,C 180,E1 -4002.787,E2 -4002.787} C_VEL
LIN {X 0,Y 538.014,Z 317.093,A -85,B 0,C 180,E1 -4005.927,E2 -4005.927} C_VEL
LIN {X 0,Y 538.043,Z 317.088,A -85,B 0,C 180,E1 -4009.225,E2 -4009.225} C_VEL
LIN {X 0,Y 537.988,Z 317.094,A -85,B 0,C 180,E1 -4012.123,E2 -4012.123} C_VEL
LIN {X 0,Y 538.008,Z 317.092,A -85,B 0,C 180,E1 -4014.918,E2 -4014.918} C_VEL
LIN {X 0,Y 538.023,Z 317.094,A -85,B 0,C 180,E1 -4017.619,E2 -4017.619} C_VEL
LIN {X 0,Y 538.014,Z 317.089,A -85,B 0,C 180,E1 -4020.24,E2 -4020.24} C_VEL
LIN {X 0,Y 538.054,Z 317.087,A -85,B 0,C 180,E1 -4022.797,E2 -4022.797} C_VEL
LIN {X 0,Y 538.07,Z 317.236,A -85,B 0,C 180,E1 -4024.468,E2 -4024.468} C_VEL
LIN {X 0,Y 539.829,Z 326.184,A -85,B 0,C 180,E1 -4025.84,E2 -4025.84} C_VEL
LIN {X 0,Y 539.381,Z 345.791,A -85,B 0,C 180,E1 -4028.603,E2 -4028.603} C_VEL
LIN {X 0,Y 538.929,Z 367.198,A -85,B 0,C 180,E1 -4031.565,E2 -4031.565} C_VEL
LIN {X 0,Y 538.856,Z 371.248,A -85,B 0,C 180,E1 -4032.122,E2 -4032.122} C_VEL
LIN {X 0,Y 540.694,Z 381.751,A -85,B 0,C 180,E1 -4032.328,E2 -4032.328} C_VEL
LIN {X 0,Y 540.113,Z 509.668,A -85,B 0,C 180,E1 -4034.07,E2 -4034.07} C_VEL
LIN {X 0,Y 539.866,Z 523.882,A -85,B 0,C 180,E1 -4034.416,E2 -4034.416} C_VEL
LIN {X 0,Y 539.662,Z 537.534,A -85,B 0,C 180,E1 -4034.903,E2 -4034.903} C_VEL
LIN {X 0,Y 539.356,Z 551.503,A -85,B 0,C 180,E1 -4035.57,E2 -4035.57} C_VEL
LIN {X 0,Y 539.014,Z 564.003,A -85,B 0,C 180,E1 -4036.331,E2 -4036.331} C_VEL
LIN {X 0,Y 538.687,Z 576.606,A -85,B 0,C 180,E1 -4037.282,E2 -4037.282} C_VEL
LIN {X 0,Y 538.429,Z 586.847,A -85,B 0,C 180,E1 -4038.226,E2 -4038.226} C_VEL
LIN {X 0,Y 538.203,Z 596.336,A -85,B 0,C 180,E1 -4039.276,E2 -4039.276} C_VEL
LIN {X 0,Y 537.969,Z 604.911,A -85,B 0,C 180,E1 -4040.412,E2 -4040.412} C_VEL
LIN {X 0,Y 537.804,Z 613.12,A -85,B 0,C 180,E1 -4041.735,E2 -4041.735} C_VEL
LIN {X 0,Y 537.66,Z 618.864,A -85,B 0,C 180,E1 -4042.867,E2 -4042.867} C_VEL
LIN {X 0,Y 537.654,Z 624.961,A -85,B 0,C 180,E1 -4044.374,E2 -4044.374} C_VEL
LIN {X 0,Y 537.55,Z 628.444,A -85,B 0,C 180,E1 -4045.501,E2 -4045.501} C_VEL
LIN {X 0,Y 537.547,Z 631.833,A -85,B 0,C 180,E1 -4047.002,E2 -4047.002} C_VEL
LIN {X 0,Y 537.447,Z 633.835,A -85,B 0,C 180,E1 -4048.501,E2 -4048.501} C_VEL
LIN {X 0,Y 537.44,Z 634.5,A -85,B 0,C 180,E1 -4050,E2 -4050} C_VEL
LIN {X 0,Y 537.447,Z 633.836,A -85,B 0,C 180,E1 -4051.499,E2 -4051.499} C_VEL
LIN {X 0,Y 537.547,Z 631.836,A -85,B 0,C 180,E1 -4052.998,E2 -4052.998} C_VEL
LIN {X 0,Y 537.55,Z 628.447,A -85,B 0,C 180,E1 -4054.499,E2 -4054.499} C_VEL
LIN {X 0,Y 537.647,Z 623.568,A -85,B 0,C 180,E1 -4056.002,E2 -4056.002} C_VEL
LIN {X 0,Y 537.704,Z 617.055,A -85,B 0,C 180,E1 -4057.51,E2 -4057.51} C_VEL
LIN {X 0,Y 537.859,Z 609.805,A -85,B 0,C 180,E1 -4058.831,E2 -4058.831} C_VEL
LIN {X 0,Y 538.063,Z 600.823,A -85,B 0,C 180,E1 -4060.156,E2 -4060.156} C_VEL
LIN {X 0,Y 538.342,Z 591.395,A -85,B 0,C 180,E1 -4061.293,E2 -4061.293} C_VEL
LIN {X 0,Y 538.564,Z 580.924,A -85,B 0,C 180,E1 -4062.338,E2 -4062.338} C_VEL
LIN {X 0,Y 538.85,Z 569.35,A -85,B 0,C 180,E1 -4063.289,E2 -4063.289} C_VEL
LIN {X 0,Y 539.183,Z 556.514,A -85,B 0,C 180,E1 -4064.146,E2 -4064.146} C_VEL
LIN {X 0,Y 539.504,Z 543.983,A -85,B 0,C 180,E1 -4064.812,E2 -4064.812} C_VEL
LIN {X 0,Y 539.785,Z 529.911,A -85,B 0,C 180,E1 -4065.388,E2 -4065.388} C_VEL
LIN {X 0,Y 540.022,Z 515.357,A -85,B 0,C 180,E1 -4065.812,E2 -4065.812} C_VEL
LIN {X 0,Y 540.141,Z 500.592,A -85,B 0,C 180,E1 -4066.075,E2 -4066.075} C_VEL
LIN {X 0,Y 540.604,Z 381.101,A -85,B 0,C 180,E1 -4067.684,E2 -4067.684} C_VEL
LIN {X 0,Y 538.859,Z 371.08,A -85,B 0,C 180,E1 -4067.9,E2 -4067.9} C_VEL
LIN {X 0,Y 539.32,Z 348.635,A -85,B 0,C 180,E1 -4070.999,E2 -4070.999} C_VEL
LIN {X 0,Y 539.817,Z 327.4,A -85,B 0,C 180,E1 -4073.983,E2 -4073.983} C_VEL
LIN {X 0,Y 539.341,Z 322.939,A -85,B 0,C 180,E1 -4074.643,E2 -4074.643} C_VEL
LIN {X 0,Y 538.059,Z 317.089,A -85,B 0,C 180,E1 -4075.564,E2 -4075.564} C_VEL
LIN {X 0,Y 538.038,Z 317.089,A -85,B 0,C 180,E1 -4078.049,E2 -4078.049} C_VEL
LIN {X 0,Y 538.017,Z 317.096,A -85,B 0,C 180,E1 -4080.626,E2 -4080.626} C_VEL
LIN {X 0,Y 538.042,Z 317.086,A -85,B 0,C 180,E1 -4083.282,E2 -4083.282} C_VEL
LIN {X 0,Y 538.02,Z 317.09,A -85,B 0,C 180,E1 -4086.001,E2 -4086.001} C_VEL
LIN {X 0,Y 538.007,Z 317.091,A -85,B 0,C 180,E1 -4088.83,E2 -4088.83} C_VEL
LIN {X 0,Y 538.029,Z 317.085,A -85,B 0,C 180,E1 -4091.772,E2 -4091.772} C_VEL
LIN {X 0,Y 538.024,Z 317.086,A -85,B 0,C 180,E1 -4094.859,E2 -4094.859} C_VEL
LIN {X 0,Y 538.026,Z 317.093,A -85,B 0,C 180,E1 -4098.12,E2 -4098.12} C_VEL
LIN {X 0,Y 538.024,Z 317.092,A -85,B 0,C 180,E1 -4100.414,E2 -4100.414} C_VEL
LIN {X 0,Y 538.017,Z 317.087,A -85,B 0,C 180,E1 -4103.067,E2 -4103.067} C_VEL
LIN {X 0,Y 538.01,Z 317.093,A -85,B 0,C 180,E1 -4105.826,E2 -4105.826} C_VEL
LIN {X 0,Y 537.997,Z 317.089,A -85,B 0,C 180,E1 -4108.498,E2 -4108.498} C_VEL
LIN {X 0,Y 538.006,Z 317.084,A -85,B 0,C 180,E1 -4111.097,E2 -4111.097} C_VEL
LIN {X 0,Y 538.01,Z 317.093,A -85,B 0,C 180,E1 -4113.632,E2 -4113.632} C_VEL
LIN {X 0,Y 537.994,Z 317.095,A -85,B 0,C 180,E1 -4116.122,E2 -4116.122} C_VEL
LIN {X 0,Y 538.023,Z 317.089,A -85,B 0,C 180,E1 -4119.348,E2 -4119.348} C_VEL
LIN {X 0,Y 538.023,Z 317.087,A -85,B 0,C 180,E1 -4122.467,E2 -4122.467} C_VEL
LIN {X 0,Y 538.036,Z 317.093,A -85,B 0,C 180,E1 -4125.63,E2 -4125.63} C_VEL
LIN {X 0,Y 538.012,Z 317.086,A -85,B 0,C 180,E1 -4128.7,E2 -4128.7} C_VEL
LIN {X 0,Y 538.018,Z 317.092,A -85,B 0,C 180,E1 -4131.739,E2 -4131.739} C_VEL
LIN {X 0,Y 538.132,Z 317.073,A -85,B 0,C 180,E1 -4134.755,E2 -4134.755} C_VEL
LIN {X 0,Y 538.141,Z 317.074,A -85,B 0,C 180,E1 -4137.755,E2 -4137.755} C_VEL
LIN {X 0,Y 538.136,Z 317.074,A -85,B 0,C 180,E1 -4140,E2 -4140} C_VEL
LIN {X 0,Y 538.115,Z 317.078,A -85,B 0,C 180,E1 -4142.995,E2 -4142.995} C_VEL
LIN {X 0,Y 538.077,Z 317.08,A -85,B 0,C 180,E1 -4145.998,E2 -4145.998} C_VEL
LIN {X 0,Y 538.043,Z 317.083,A -85,B 0,C 180,E1 -4148.261,E2 -4148.261} C_VEL
LIN {X 0,Y 538.07,Z 317.081,A -85,B 0,C 180,E1 -4151.597,E2 -4151.597} C_VEL
LIN {X 0,Y 538.043,Z 317.09,A -85,B 0,C 180,E1 -4154.856,E2 -4154.856} C_VEL
LIN {X 0,Y 538.024,Z 317.089,A -85,B 0,C 180,E1 -4157.533,E2 -4157.533} C_VEL
LIN {X 0,Y 538.025,Z 317.09,A -85,B 0,C 180,E1 -4160.652,E2 -4160.652} C_VEL
LIN {X 0,Y 537.992,Z 317.09,A -85,B 0,C 180,E1 -4163.889,E2 -4163.889} C_VEL
LIN {X 0,Y 538.032,Z 317.088,A -85,B 0,C 180,E1 -4166.368,E2 -4166.368} C_VEL
LIN {X 0,Y 538.021,Z 317.094,A -85,B 0,C 180,E1 -4168.934,E2 -4168.934} C_VEL
LIN {X 0,Y 538.006,Z 317.088,A -85,B 0,C 180,E1 -4171.889,E2 -4171.889} C_VEL
LIN {X 0,Y 538.015,Z 317.095,A -85,B 0,C 180,E1 -4174.62,E2 -4174.62} C_VEL
LIN {X 0,Y 537.997,Z 317.09,A -85,B 0,C 180,E1 -4177.171,E2 -4177.171} C_VEL
LIN {X 0,Y 538.017,Z 317.088,A -85,B 0,C 180,E1 -4180.232,E2 -4180.232} C_VEL
LIN {X 0,Y 537.367,Z 317.174,A -85,B 0,C 180,E1 -4180.857,E2 -4180.857} C_VEL
LIN {X 0,Y 534.519,Z 317.527,A -85,B 0,C 180,E1 -4181.872,E2 -4181.872} C_VEL
LIN {X 0,Y 532.096,Z 317.832,A -85,B 0,C 180,E1 -4182.689,E2 -4182.689} C_VEL
LIN {X 0,Y 531.048,Z 317.957,A -85,B 0,C 180,E1 -4183.32,E2 -4183.32} C_VEL
LIN {X 0,Y 530.959,Z 317.967,A -85,B 0,C 180,E1 -4183.534,E2 -4183.534} C_VEL
LIN {X 0,Y 530.951,Z 317.975,A -85,B 0,C 180,E1 -4186.506,E2 -4186.506} C_VEL
LIN {X 0,Y 530.984,Z 317.966,A -85,B 0,C 180,E1 -4188.977,E2 -4188.977} C_VEL
LIN {X 0,Y 530.957,Z 317.968,A -85,B 0,C 180,E1 -4191.531,E2 -4191.531} C_VEL
LIN {X 0,Y 530.978,Z 317.97,A -85,B 0,C 180,E1 -4194.383,E2 -4194.383} C_VEL
LIN {X 0,Y 530.971,Z 317.968,A -85,B 0,C 180,E1 -4197.135,E2 -4197.135} C_VEL
LIN {X 0,Y 530.971,Z 317.972,A -85,B 0,C 180,E1 -4199.804,E2 -4199.804} C_VEL
LIN {X 0,Y 531.045,Z 317.969,A -85,B 0,C 180,E1 -4201.6,E2 -4201.6} C_VEL
LIN {X 0,Y 532.197,Z 325.257,A -85,B 0,C 180,E1 -4202.898,E2 -4202.898} C_VEL
LIN {X 0,Y 531.868,Z 340.199,A -85,B 0,C 180,E1 -4205.404,E2 -4205.404} C_VEL
LIN {X 0,Y 531.795,Z 343.39,A -85,B 0,C 180,E1 -4205.934,E2 -4205.934} C_VEL
LIN {X 0,Y 533.975,Z 354.855,A -85,B 0,C 180,E1 -4206.172,E2 -4206.172} C_VEL
LIN {X 0,Y 533.304,Z 479.575,A -85,B 0,C 180,E1 -4207.89,E2 -4207.89} C_VEL
LIN {X 0,Y 533.109,Z 493.883,A -85,B 0,C 180,E1 -4208.237,E2 -4208.237} C_VEL
LIN {X 0,Y 532.843,Z 507.755,A -85,B 0,C 180,E1 -4208.734,E2 -4208.734} C_VEL
LIN {X 0,Y 532.514,Z 520.825,A -85,B 0,C 180,E1 -4209.358,E2 -4209.358} C_VEL
LIN {X 0,Y 532.139,Z 533.352,A -85,B 0,C 180,E1 -4210.119,E2 -4210.119} C_VEL
LIN {X 0,Y 531.814,Z 545.167,A -85,B 0,C 180,E1 -4211.009,E2 -4211.009} C_VEL
LIN {X 0,Y 531.519,Z 555.336,A -85,B 0,C 180,E1 -4211.937,E2 -4211.937} C_VEL
LIN {X 0,Y 531.183,Z 565.73,A -85,B 0,C 180,E1 -4213.078,E2 -4213.078} C_VEL
LIN {X 0,Y 530.932,Z 574.581,A -85,B 0,C 180,E1 -4214.255,E2 -4214.255} C_VEL
LIN {X 0,Y 530.731,Z 583.014,A -85,B 0,C 180,E1 -4215.624,E2 -4215.624} C_VEL
LIN {X 0,Y 530.605,Z 589.729,A -85,B 0,C 180,E1 -4216.988,E2 -4216.988} C_VEL
LIN {X 0,Y 530.504,Z 595.648,A -85,B 0,C 180,E1 -4218.538,E2 -4218.538} C_VEL
LIN {X 0,Y 530.423,Z 599.954,A -85,B 0,C 180,E1 -4220.082,E2 -4220.082} C_VEL
LIN {X 0,Y 530.42,Z 602.788,A -85,B 0,C 180,E1 -4221.62,E2 -4221.62} C_VEL
LIN {X 0,Y 530.468,Z 604.252,A -85,B 0,C 180,E1 -4223.152,E2 -4223.152} C_VEL
LIN {X 0,Y 530.444,Z 604.373,A -85,B 0,C 180,E1 -4224.679,E2 -4224.679} C_VEL
LIN {X 0,Y 530.479,Z 603.162,A -85,B 0,C 180,E1 -4226.202,E2 -4226.202} C_VEL
LIN {X 0,Y 530.412,Z 600.615,A -85,B 0,C 180,E1 -4227.722,E2 -4227.722} C_VEL
LIN {X 0,Y 530.415,Z 596.656,A -85,B 0,C 180,E1 -4229.241,E2 -4229.241} C_VEL
LIN {X 0,Y 530.487,Z 591.177,A -85,B 0,C 180,E1 -4230.759,E2 -4230.759} C_VEL
LIN {X 0,Y 530.69,Z 585.989,A -85,B 0,C 180,E1 -4231.897,E2 -4231.897} C_VEL
LIN {X 0,Y 530.79,Z 578.551,A -85,B 0,C 180,E1 -4233.226,E2 -4233.226} C_VEL
LIN {X 0,Y 531.09,Z 570.811,A -85,B 0,C 180,E1 -4234.364,E2 -4234.364} C_VEL
LIN {X 0,Y 531.335,Z 561.512,A -85,B 0,C 180,E1 -4235.503,E2 -4235.503} C_VEL
LIN {X 0,Y 531.669,Z 550.196,A -85,B 0,C 180,E1 -4236.642,E2 -4236.642} C_VEL
LIN {X 0,Y 531.982,Z 538.683,A -85,B 0,C 180,E1 -4237.591,E2 -4237.591} C_VEL
LIN {X 0,Y 532.405,Z 525.892,A -85,B 0,C 180,E1 -4238.444,E2 -4238.444} C_VEL
LIN {X 0,Y 532.756,Z 512.391,A -85,B 0,C 180,E1 -4239.156,E2 -4239.156} C_VEL
LIN {X 0,Y 533.012,Z 498.65,A -85,B 0,C 180,E1 -4239.702,E2 -4239.702} C_VEL
LIN {X 0,Y 533.274,Z 485.211,A -85,B 0,C 180,E1 -4240.08,E2 -4240.08} C_VEL
LIN {X 0,Y 533.392,Z 470.355,A -85,B 0,C 180,E1 -4240.342,E2 -4240.342} C_VEL
LIN {X 0,Y 533.865,Z 353.55,A -85,B 0,C 180,E1 -4241.939,E2 -4241.939} C_VEL
LIN {X 0,Y 531.782,Z 343.335,A -85,B 0,C 180,E1 -4242.162,E2 -4242.162} C_VEL
LIN {X 0,Y 532.19,Z 326.861,A -85,B 0,C 180,E1 -4244.916,E2 -4244.916} C_VEL
LIN {X 0,Y 531.885,Z 322.467,A -85,B 0,C 180,E1 -4245.676,E2 -4245.676} C_VEL
LIN {X 0,Y 531.018,Z 317.966,A -85,B 0,C 180,E1 -4246.507,E2 -4246.507} C_VEL
LIN {X 0,Y 530.998,Z 317.967,A -85,B 0,C 180,E1 -4249.322,E2 -4249.322} C_VEL
LIN {X 0,Y 530.981,Z 317.97,A -85,B 0,C 180,E1 -4252.101,E2 -4252.101} C_VEL
LIN {X 0,Y 530.997,Z 317.963,A -85,B 0,C 180,E1 -4255.057,E2 -4255.057} C_VEL
LIN {X 0,Y 531.017,Z 317.967,A -85,B 0,C 180,E1 -4257.594,E2 -4257.594} C_VEL
LIN {X 0,Y 530.975,Z 317.965,A -85,B 0,C 180,E1 -4260.644,E2 -4260.644} C_VEL
LIN {X 0,Y 530.991,Z 317.97,A -85,B 0,C 180,E1 -4263.771,E2 -4263.771} C_VEL
LIN {X 0,Y 530.965,Z 317.965,A -85,B 0,C 180,E1 -4266.556,E2 -4266.556} C_VEL
LIN {X 0,Y 530.978,Z 317.963,A -85,B 0,C 180,E1 -4269.853,E2 -4269.853} C_VEL
LIN {X 0,Y 530.974,Z 317.964,A -85,B 0,C 180,E1 -4272.456,E2 -4272.456} C_VEL
LIN {X 0,Y 530.984,Z 317.97,A -85,B 0,C 180,E1 -4275.62,E2 -4275.62} C_VEL
LIN {X 0,Y 530.988,Z 317.962,A -85,B 0,C 180,E1 -4278.563,E2 -4278.563} C_VEL
LIN {X 0,Y 530.95,Z 317.971,A -85,B 0,C 180,E1 -4281.528,E2 -4281.528} C_VEL
LIN {X 0,Y 530.948,Z 317.968,A -85,B 0,C 180,E1 -4284.379,E2 -4284.379} C_VEL
LIN {X 0,Y 530.958,Z 317.973,A -85,B 0,C 180,E1 -4287.132,E2 -4287.132} C_VEL
LIN {X 0,Y 530.959,Z 317.967,A -85,B 0,C 180,E1 -4289.802,E2 -4289.802} C_VEL
LIN {X 0,Y 531.001,Z 317.959,A -85,B 0,C 180,E1 -4292.467,E2 -4292.467} C_VEL
LIN {X 0,Y 530.958,Z 317.973,A -85,B 0,C 180,E1 -4294.94,E2 -4294.94} C_VEL
LIN {X 0,Y 530.965,Z 317.964,A -85,B 0,C 180,E1 -4297.897,E2 -4297.897} C_VEL
LIN {X 0,Y 530.971,Z 317.965,A -85,B 0,C 180,E1 -4300.676,E2 -4300.676} C_VEL
LIN {X 0,Y 530.951,Z 317.974,A -85,B 0,C 180,E1 -4303.069,E2 -4303.069} C_VEL
LIN {X 0,Y 531,Z 317.96,A -85,B 0,C 180,E1 -4305.435,E2 -4305.435} C_VEL
LIN {X 0,Y 531.017,Z 317.96,A -85,B 0,C 180,E1 -4308.549,E2 -4308.549} C_VEL
LIN {X 0,Y 531.017,Z 317.959,A -85,B 0,C 180,E1 -4311.629,E2 -4311.629} C_VEL
LIN {X 0,Y 531.089,Z 317.953,A -85,B 0,C 180,E1 -4314.685,E2 -4314.685} C_VEL
LIN {X 0,Y 531.111,Z 317.946,A -85,B 0,C 180,E1 -4317.725,E2 -4317.725} C_VEL
LIN {X 0,Y 531.134,Z 317.949,A -85,B 0,C 180,E1 -4320.758,E2 -4320.758} C_VEL
LIN {X 0,Y 531.043,Z 317.955,A -85,B 0,C 180,E1 -4323.034,E2 -4323.034} C_VEL
LIN {X 0,Y 531.026,Z 317.962,A -85,B 0,C 180,E1 -4326.078,E2 -4326.078} C_VEL
LIN {X 0,Y 530.991,Z 317.959,A -85,B 0,C 180,E1 -4329.139,E2 -4329.139} C_VEL
LIN {X 0,Y 531.034,Z 317.958,A -85,B 0,C 180,E1 -4331.67,E2 -4331.67} C_VEL
LIN {X 0,Y 531.017,Z 317.957,A -85,B 0,C 180,E1 -4334.956,E2 -4334.956} C_VEL
LIN {X 0,Y 530.966,Z 317.967,A -85,B 0,C 180,E1 -4337.724,E2 -4337.724} C_VEL
LIN {X 0,Y 531.011,Z 317.967,A -85,B 0,C 180,E1 -4340.128,E2 -4340.128} C_VEL
LIN {X 0,Y 530.931,Z 317.972,A -85,B 0,C 180,E1 -4342.574,E2 -4342.574} C_VEL
LIN {X 0,Y 530.975,Z 317.963,A -85,B 0,C 180,E1 -4345.059,E2 -4345.059} C_VEL
LIN {X 0,Y 530.957,Z 317.969,A -85,B 0,C 180,E1 -4347.599,E2 -4347.599} C_VEL
LIN {X 0,Y 530.957,Z 317.971,A -85,B 0,C 180,E1 -4350.198,E2 -4350.198} C_VEL
LIN {X 0,Y 530.956,Z 317.967,A -85,B 0,C 180,E1 -4352.867,E2 -4352.867} C_VEL
LIN {X 0,Y 530.964,Z 317.971,A -85,B 0,C 180,E1 -4355.619,E2 -4355.619} C_VEL
LIN {X 0,Y 530.956,Z 317.967,A -85,B 0,C 180,E1 -4358.654,E2 -4358.654} C_VEL
LIN {X 0,Y 530.989,Z 317.965,A -85,B 0,C 180,E1 -4361.436,E2 -4361.436} C_VEL
LIN {X 0,Y 530.979,Z 317.964,A -85,B 0,C 180,E1 -4364.548,E2 -4364.548} C_VEL
LIN {X 0,Y 530.978,Z 317.971,A -85,B 0,C 180,E1 -4367.835,E2 -4367.835} C_VEL
LIN {X 0,Y 530.98,Z 317.965,A -85,B 0,C 180,E1 -4370.557,E2 -4370.557} C_VEL
LIN {X 0,Y 530.964,Z 317.976,A -85,B 0,C 180,E1 -4373.443,E2 -4373.443} C_VEL
LIN {X 0,Y 530.996,Z 317.964,A -85,B 0,C 180,E1 -4376.495,E2 -4376.495} C_VEL
LIN {X 0,Y 530.971,Z 317.974,A -85,B 0,C 180,E1 -4379.356,E2 -4379.356} C_VEL
LIN {X 0,Y 531.01,Z 317.963,A -85,B 0,C 180,E1 -4382.468,E2 -4382.468} C_VEL
LIN {X 0,Y 531.017,Z 317.983,A -85,B 0,C 180,E1 -4384.239,E2 -4384.239} C_VEL
LIN {X 0,Y 532.9,Z 327.141,A -85,B 0,C 180,E1 -4385.67,E2 -4385.67} C_VEL
LIN {X 0,Y 532.555,Z 342.761,A -85,B 0,C 180,E1 -4387.908,E2 -4387.908} C_VEL
LIN {X 0,Y 532.114,Z 362.725,A -85,B 0,C 180,E1 -4390.72,E2 -4390.72} C_VEL
LIN {X 0,Y 531.893,Z 371.022,A -85,B 0,C 180,E1 -4391.877,E2 -4391.877} C_VEL
LIN {X 0,Y 533.916,Z 383.655,A -85,B 0,C 180,E1 -4392.125,E2 -4392.125} C_VEL
LIN {X 0,Y 533.281,Z 509.455,A -85,B 0,C 180,E1 -4393.86,E2 -4393.86} C_VEL
LIN {X 0,Y 533.008,Z 524.031,A -85,B 0,C 180,E1 -4394.222,E2 -4394.222} C_VEL
LIN {X 0,Y 532.75,Z 538.459,A -85,B 0,C 180,E1 -4394.751,E2 -4394.751} C_VEL
LIN {X 0,Y 532.449,Z 551.297,A -85,B 0,C 180,E1 -4395.379,E2 -4395.379} C_VEL
LIN {X 0,Y 532.065,Z 563.798,A -85,B 0,C 180,E1 -4396.149,E2 -4396.149} C_VEL
LIN {X 0,Y 531.712,Z 576.402,A -85,B 0,C 180,E1 -4397.112,E2 -4397.112} C_VEL
LIN {X 0,Y 531.42,Z 587.323,A -85,B 0,C 180,E1 -4398.138,E2 -4398.138} C_VEL
LIN {X 0,Y 531.129,Z 597.707,A -85,B 0,C 180,E1 -4399.325,E2 -4399.325} C_VEL
LIN {X 0,Y 530.9,Z 606.076,A -85,B 0,C 180,E1 -4400.476,E2 -4400.476} C_VEL
LIN {X 0,Y 530.709,Z 614.077,A -85,B 0,C 180,E1 -4401.816,E2 -4401.816} C_VEL
LIN {X 0,Y 530.573,Z 620.521,A -85,B 0,C 180,E1 -4403.153,E2 -4403.153} C_VEL
LIN {X 0,Y 530.584,Z 624.961,A -85,B 0,C 180,E1 -4404.299,E2 -4404.299} C_VEL
LIN {X 0,Y 530.449,Z 628.444,A -85,B 0,C 180,E1 -4405.441,E2 -4405.441} C_VEL
LIN {X 0,Y 530.452,Z 631.832,A -85,B 0,C 180,E1 -4406.962,E2 -4406.962} C_VEL
LIN {X 0,Y 530.357,Z 633.835,A -85,B 0,C 180,E1 -4408.481,E2 -4408.481} C_VEL
LIN {X 0,Y 530.341,Z 634.5,A -85,B 0,C 180,E1 -4410,E2 -4410} C_VEL
LIN {X 0,Y 530.357,Z 633.837,A -85,B 0,C 180,E1 -4411.519,E2 -4411.519} C_VEL
LIN {X 0,Y 530.452,Z 631.836,A -85,B 0,C 180,E1 -4413.038,E2 -4413.038} C_VEL
LIN {X 0,Y 530.449,Z 628.447,A -85,B 0,C 180,E1 -4414.559,E2 -4414.559} C_VEL
LIN {X 0,Y 530.56,Z 623.568,A -85,B 0,C 180,E1 -4416.083,E2 -4416.083} C_VEL
LIN {X 0,Y 530.585,Z 618.842,A -85,B 0,C 180,E1 -4417.229,E2 -4417.229} C_VEL
LIN {X 0,Y 530.756,Z 611.971,A -85,B 0,C 180,E1 -4418.567,E2 -4418.567} C_VEL
LIN {X 0,Y 530.927,Z 603.439,A -85,B 0,C 180,E1 -4419.909,E2 -4419.909} C_VEL
LIN {X 0,Y 531.223,Z 594.541,A -85,B 0,C 180,E1 -4421.059,E2 -4421.059} C_VEL
LIN {X 0,Y 531.488,Z 583.763,A -85,B 0,C 180,E1 -4422.214,E2 -4422.214} C_VEL
LIN {X 0,Y 531.812,Z 571.682,A -85,B 0,C 180,E1 -4423.274,E2 -4423.274} C_VEL
LIN {X 0,Y 532.177,Z 559.473,A -85,B 0,C 180,E1 -4424.141,E2 -4424.141} C_VEL
LIN {X 0,Y 532.53,Z 547.735,A -85,B 0,C 180,E1 -4424.815,E2 -4424.815} C_VEL
LIN {X 0,Y 532.881,Z 534.204,A -85,B 0,C 180,E1 -4425.423,E2 -4425.423} C_VEL
LIN {X 0,Y 533.047,Z 520.611,A -85,B 0,C 180,E1 -4425.879,E2 -4425.879} C_VEL
LIN {X 0,Y 533.298,Z 506.676,A -85,B 0,C 180,E1 -4426.188,E2 -4426.188} C_VEL
LIN {X 0,Y 533.91,Z 382.646,A -85,B 0,C 180,E1 -4427.889,E2 -4427.889} C_VEL
LIN {X 0,Y 531.896,Z 370.991,A -85,B 0,C 180,E1 -4428.125,E2 -4428.125} C_VEL
LIN {X 0,Y 532.415,Z 348.429,A -85,B 0,C 180,E1 -4431.284,E2 -4431.284} C_VEL
LIN {X 0,Y 532.951,Z 328.476,A -85,B 0,C 180,E1 -4434.128,E2 -4434.128} C_VEL
LIN {X 0,Y 532.307,Z 323.842,A -85,B 0,C 180,E1 -4434.833,E2 -4434.833} C_VEL
LIN {X 0,Y 531.017,Z 317.967,A -85,B 0,C 180,E1 -4435.761,E2 -4435.761} C_VEL
LIN {X 0,Y 530.994,Z 317.969,A -85,B 0,C 180,E1 -4438.455,E2 -4438.455} C_VEL
LIN {X 0,Y 530.954,Z 317.972,A -85,B 0,C 180,E1 -4441.078,E2 -4441.078} C_VEL
LIN {X 0,Y 530.985,Z 317.966,A -85,B 0,C 180,E1 -4443.772,E2 -4443.772} C_VEL
LIN {X 0,Y 530.964,Z 317.97,A -85,B 0,C 180,E1 -4446.557,E2 -4446.557} C_VEL
LIN {X 0,Y 530.972,Z 317.966,A -85,B 0,C 180,E1 -4449.853,E2 -4449.853} C_VEL
LIN {X 0,Y 530.973,Z 317.97,A -85,B 0,C 180,E1 -4452.456,E2 -4452.456} C_VEL
LIN {X 0,Y 530.978,Z 317.963,A -85,B 0,C 180,E1 -4455.62,E2 -4455.62} C_VEL
LIN {X 0,Y 530.989,Z 317.967,A -85,B 0,C 180,E1 -4458.564,E2 -4458.564} C_VEL
LIN {X 0,Y 530.947,Z 317.97,A -85,B 0,C 180,E1 -4461.529,E2 -4461.529} C_VEL
LIN {X 0,Y 530.964,Z 317.97,A -85,B 0,C 180,E1 -4464.381,E2 -4464.381} C_VEL
LIN {X 0,Y 530.956,Z 317.967,A -85,B 0,C 180,E1 -4467.133,E2 -4467.133} C_VEL
LIN {X 0,Y 530.957,Z 317.968,A -85,B 0,C 180,E1 -4469.802,E2 -4469.802} C_VEL
LIN {X 0,Y 530.955,Z 317.969,A -85,B 0,C 180,E1 -4472.477,E2 -4472.477} C_VEL
LIN {X 0,Y 530.975,Z 317.963,A -85,B 0,C 180,E1 -4474.941,E2 -4474.941} C_VEL
LIN {X 0,Y 530.958,Z 317.969,A -85,B 0,C 180,E1 -4478.246,E2 -4478.246} C_VEL
LIN {X 0,Y 530.968,Z 317.965,A -85,B 0,C 180,E1 -4480.676,E2 -4480.676} C_VEL
LIN {X 0,Y 530.949,Z 317.969,A -85,B 0,C 180,E1 -4483.07,E2 -4483.07} C_VEL
LIN {X 0,Y 530.993,Z 317.967,A -85,B 0,C 180,E1 -4485.435,E2 -4485.435} C_VEL
LIN {X 0,Y 530.974,Z 317.962,A -85,B 0,C 180,E1 -4488.549,E2 -4488.549} C_VEL
LIN {X 0,Y 530.966,Z 317.972,A -85,B 0,C 180,E1 -4491.628,E2 -4491.628} C_VEL
LIN {X 0,Y 531.09,Z 317.95,A -85,B 0,C 180,E1 -4494.685,E2 -4494.685} C_VEL
LIN {X 0,Y 531.114,Z 317.95,A -85,B 0,C 180,E1 -4497.725,E2 -4497.725} C_VEL
LIN {X 0,Y 531.106,Z 317.95,A -85,B 0,C 180,E1 -4500,E2 -4500} C_VEL
LIN {X 0,Y 531.083,Z 317.954,A -85,B 0,C 180,E1 -4503.035,E2 -4503.035} C_VEL
LIN {X 0,Y 531.036,Z 317.957,A -85,B 0,C 180,E1 -4506.078,E2 -4506.078} C_VEL
LIN {X 0,Y 530.996,Z 317.969,A -85,B 0,C 180,E1 -4509.139,E2 -4509.139} C_VEL
LIN {X 0,Y 531.014,Z 317.957,A -85,B 0,C 180,E1 -4512.226,E2 -4512.226} C_VEL
LIN {X 0,Y 530.981,Z 317.967,A -85,B 0,C 180,E1 -4515.351,E2 -4515.351} C_VEL
LIN {X 0,Y 530.972,Z 317.968,A -85,B 0,C 180,E1 -4518.522,E2 -4518.522} C_VEL
LIN {X 0,Y 530.987,Z 317.97,A -85,B 0,C 180,E1 -4520.939,E2 -4520.939} C_VEL
LIN {X 0,Y 530.961,Z 317.967,A -85,B 0,C 180,E1 -4524.226,E2 -4524.226} C_VEL
LIN {X 0,Y 530.992,Z 317.971,A -85,B 0,C 180,E1 -4526.745,E2 -4526.745} C_VEL
LIN {X 0,Y 530.972,Z 317.967,A -85,B 0,C 180,E1 -4529.324,E2 -4529.324} C_VEL
LIN {X 0,Y 530.963,Z 317.966,A -85,B 0,C 180,E1 -4532.102,E2 -4532.102} C_VEL
LIN {X 0,Y 530.97,Z 317.971,A -85,B 0,C 180,E1 -4534.853,E2 -4534.853} C_VEL
LIN {X 0,Y 530.959,Z 317.965,A -85,B 0,C 180,E1 -4537.509,E2 -4537.509} C_VEL
LIN {X 0,Y 530.981,Z 317.97,A -85,B 0,C 180,E1 -4540.434,E2 -4540.434} C_VEL
LIN {X 0,Y 530.961,Z 317.967,A -85,B 0,C 180,E1 -4543.496,E2 -4543.496} C_VEL
LIN {X 0,Y 530.959,Z 317.967,A -85,B 0,C 180,E1 -4543.534,E2 -4543.534} C_VEL
LIN {X 0,Y 530.284,Z 318.057,A -85,B 0,C 180,E1 -4544.167,E2 -4544.167} C_VEL
LIN {X 0,Y 527.435,Z 318.413,A -85,B 0,C 180,E1 -4545.196,E2 -4545.196} C_VEL
LIN {X 0,Y 525.031,Z 318.714,A -85,B 0,C 180,E1 -4546.024,E2 -4546.024} C_VEL
LIN {X 0,Y 523.997,Z 318.84,A -85,B 0,C 180,E1 -4546.663,E2 -4546.663} C_VEL
LIN {X 0,Y 523.912,Z 318.848,A -85,B 0,C 180,E1 -4546.88,E2 -4546.88} C_VEL
LIN {X 0,Y 523.939,Z 318.844,A -85,B 0,C 180,E1 -4548.909,E2 -4548.909} C_VEL
LIN {X 0,Y 523.915,Z 318.849,A -85,B 0,C 180,E1 -4551.899,E2 -4551.899} C_VEL
LIN {X 0,Y 523.936,Z 318.842,A -85,B 0,C 180,E1 -4554.91,E2 -4554.91} C_VEL
LIN {X 0,Y 523.938,Z 318.846,A -85,B 0,C 180,E1 -4557.68,E2 -4557.68} C_VEL
LIN {X 0,Y 523.956,Z 318.846,A -85,B 0,C 180,E1 -4560.677,E2 -4560.677} C_VEL
LIN {X 0,Y 524.003,Z 318.846,A -85,B 0,C 180,E1 -4561.404,E2 -4561.404} C_VEL
LIN {X 0,Y 525.255,Z 326.134,A -85,B 0,C 180,E1 -4562.725,E2 -4562.725} C_VEL
LIN {X 0,Y 524.943,Z 341.114,A -85,B 0,C 180,E1 -4565.268,E2 -4565.268} C_VEL
LIN {X 0,Y 524.885,Z 343.647,A -85,B 0,C 180,E1 -4565.69,E2 -4565.69} C_VEL
LIN {X 0,Y 527.235,Z 355.461,A -85,B 0,C 180,E1 -4565.942,E2 -4565.942} C_VEL
LIN {X 0,Y 526.489,Z 480.563,A -85,B 0,C 180,E1 -4567.691,E2 -4567.691} C_VEL
LIN {X 0,Y 526.282,Z 494.587,A -85,B 0,C 180,E1 -4568.043,E2 -4568.043} C_VEL
LIN {X 0,Y 525.991,Z 508.326,A -85,B 0,C 180,E1 -4568.546,E2 -4568.546} C_VEL
LIN {X 0,Y 525.637,Z 521.778,A -85,B 0,C 180,E1 -4569.203,E2 -4569.203} C_VEL
LIN {X 0,Y 525.235,Z 533.785,A -85,B 0,C 180,E1 -4569.948,E2 -4569.948} C_VEL
LIN {X 0,Y 524.872,Z 545.558,A -85,B 0,C 180,E1 -4570.85,E2 -4570.85} C_VEL
LIN {X 0,Y 524.539,Z 556.293,A -85,B 0,C 180,E1 -4571.85,E2 -4571.85} C_VEL
LIN {X 0,Y 524.161,Z 566.89,A -85,B 0,C 180,E1 -4573.045,E2 -4573.045} C_VEL
LIN {X 0,Y 523.894,Z 575.576,A -85,B 0,C 180,E1 -4574.238,E2 -4574.238} C_VEL
LIN {X 0,Y 523.67,Z 583.813,A -85,B 0,C 180,E1 -4575.625,E2 -4575.625} C_VEL
LIN {X 0,Y 523.551,Z 589.578,A -85,B 0,C 180,E1 -4576.809,E2 -4576.809} C_VEL
LIN {X 0,Y 523.433,Z 594.238,A -85,B 0,C 180,E1 -4577.988,E2 -4577.988} C_VEL
LIN {X 0,Y 523.42,Z 597.971,A -85,B 0,C 180,E1 -4579.165,E2 -4579.165} C_VEL
LIN {X 0,Y 523.281,Z 601.597,A -85,B 0,C 180,E1 -4580.726,E2 -4580.726} C_VEL
LIN {X 0,Y 523.331,Z 603.799,A -85,B 0,C 180,E1 -4582.282,E2 -4582.282} C_VEL
LIN {X 0,Y 523.37,Z 604.648,A -85,B 0,C 180,E1 -4583.833,E2 -4583.833} C_VEL
LIN {X 0,Y 523.301,Z 604.175,A -85,B 0,C 180,E1 -4585.378,E2 -4585.378} C_VEL
LIN {X 0,Y 523.399,Z 603.44,A -85,B 0,C 180,E1 -4586.15,E2 -4586.15} C_VEL
LIN {X 0,Y 523.336,Z 600.979,A -85,B 0,C 180,E1 -4587.691,E2 -4587.691} C_VEL
LIN {X 0,Y 523.33,Z 597.114,A -85,B 0,C 180,E1 -4589.231,E2 -4589.231} C_VEL
LIN {X 0,Y 523.409,Z 591.711,A -85,B 0,C 180,E1 -4590.769,E2 -4590.769} C_VEL
LIN {X 0,Y 523.632,Z 586.595,A -85,B 0,C 180,E1 -4591.923,E2 -4591.923} C_VEL
LIN {X 0,Y 523.727,Z 579.261,A -85,B 0,C 180,E1 -4593.269,E2 -4593.269} C_VEL
LIN {X 0,Y 524.063,Z 571.61,A -85,B 0,C 180,E1 -4594.422,E2 -4594.422} C_VEL
LIN {X 0,Y 524.332,Z 562.44,A -85,B 0,C 180,E1 -4595.576,E2 -4595.576} C_VEL
LIN {X 0,Y 524.687,Z 551.276,A -85,B 0,C 180,E1 -4596.731,E2 -4596.731} C_VEL
LIN {X 0,Y 525.058,Z 539.938,A -85,B 0,C 180,E1 -4597.692,E2 -4597.692} C_VEL
LIN {X 0,Y 525.483,Z 527.388,A -85,B 0,C 180,E1 -4598.557,E2 -4598.557} C_VEL
LIN {X 0,Y 525.83,Z 515.198,A -85,B 0,C 180,E1 -4599.229,E2 -4599.229} C_VEL
LIN {X 0,Y 526.16,Z 501.714,A -85,B 0,C 180,E1 -4599.805,E2 -4599.805} C_VEL
LIN {X 0,Y 526.455,Z 487.702,A -85,B 0,C 180,E1 -4600.237,E2 -4600.237} C_VEL
LIN {X 0,Y 526.58,Z 472.892,A -85,B 0,C 180,E1 -4600.526,E2 -4600.526} C_VEL
LIN {X 0,Y 527.089,Z 354.271,A -85,B 0,C 180,E1 -4602.17,E2 -4602.17} C_VEL
LIN {X 0,Y 524.856,Z 343.535,A -85,B 0,C 180,E1 -4602.411,E2 -4602.411} C_VEL
LIN {X 0,Y 525.284,Z 327.737,A -85,B 0,C 180,E1 -4605.084,E2 -4605.084} C_VEL
LIN {X 0,Y 524.791,Z 322.926,A -85,B 0,C 180,E1 -4605.934,E2 -4605.934} C_VEL
LIN {X 0,Y 523.964,Z 318.844,A -85,B 0,C 180,E1 -4606.71,E2 -4606.71} C_VEL
LIN {X 0,Y 523.978,Z 318.844,A -85,B 0,C 180,E1 -4609.591,E2 -4609.591} C_VEL
LIN {X 0,Y 523.922,Z 318.848,A -85,B 0,C 180,E1 -4612.243,E2 -4612.243} C_VEL
LIN {X 0,Y 523.95,Z 318.844,A -85,B 0,C 180,E1 -4615.418,E2 -4615.418} C_VEL
LIN {X 0,Y 523.968,Z 318.842,A -85,B 0,C 180,E1 -4617.998,E2 -4617.998} C_VEL
LIN {X 0,Y 523.946,Z 318.841,A -85,B 0,C 180,E1 -4620.854,E2 -4620.854} C_VEL
LIN {X 0,Y 523.962,Z 318.846,A -85,B 0,C 180,E1 -4623.734,E2 -4623.734} C_VEL
LIN {X 0,Y 523.919,Z 318.843,A -85,B 0,C 180,E1 -4626.403,E2 -4626.403} C_VEL
LIN {X 0,Y 523.92,Z 318.846,A -85,B 0,C 180,E1 -4629.083,E2 -4629.083} C_VEL
LIN {X 0,Y 523.948,Z 318.841,A -85,B 0,C 180,E1 -4632.118,E2 -4632.118} C_VEL
LIN {X 0,Y 523.951,Z 318.846,A -85,B 0,C 180,E1 -4635.308,E2 -4635.308} C_VEL
LIN {X 0,Y 523.95,Z 318.839,A -85,B 0,C 180,E1 -4638.689,E2 -4638.689} C_VEL
LIN {X 0,Y 523.91,Z 318.85,A -85,B 0,C 180,E1 -4641.08,E2 -4641.08} C_VEL
LIN {X 0,Y 523.893,Z 318.849,A -85,B 0,C 180,E1 -4643.824,E2 -4643.824} C_VEL
LIN {X 0,Y 523.905,Z 318.845,A -85,B 0,C 180,E1 -4646.632,E2 -4646.632} C_VEL
LIN {X 0,Y 523.947,Z 318.846,A -85,B 0,C 180,E1 -4649.355,E2 -4649.355} C_VEL
LIN {X 0,Y 523.964,Z 318.834,A -85,B 0,C 180,E1 -4652.281,E2 -4652.281} C_VEL
LIN {X 0,Y 523.901,Z 318.849,A -85,B 0,C 180,E1 -4655.426,E2 -4655.426} C_VEL
LIN {X 0,Y 523.926,Z 318.841,A -85,B 0,C 180,E1 -4657.939,E2 -4657.939} C_VEL
LIN {X 0,Y 523.957,Z 318.835,A -85,B 0,C 180,E1 -4660.407,E2 -4660.407} C_VEL
LIN {X 0,Y 523.93,Z 318.85,A -85,B 0,C 180,E1 -4662.836,E2 -4662.836} C_VEL
LIN {X 0,Y 523.96,Z 318.839,A -85,B 0,C 180,E1 -4665.235,E2 -4665.235} C_VEL
LIN {X 0,Y 524,Z 318.831,A -85,B 0,C 180,E1 -4668.394,E2 -4668.394} C_VEL
LIN {X 0,Y 523.969,Z 318.837,A -85,B 0,C 180,E1 -4671.515,E2 -4671.515} C_VEL
LIN {X 0,Y 524,Z 318.831,A -85,B 0,C 180,E1 -4673.84,E2 -4673.84} C_VEL
LIN {X 0,Y 524.021,Z 318.834,A -85,B 0,C 180,E1 -4676.925,E2 -4676.925} C_VEL
LIN {X 0,Y 523.982,Z 318.841,A -85,B 0,C 180,E1 -4678.463,E2 -4678.463} C_VEL
LIN {X 0,Y 524.104,Z 318.825,A -85,B 0,C 180,E1 -4680.768,E2 -4680.768} C_VEL
LIN {X 0,Y 523.984,Z 318.834,A -85,B 0,C 180,E1 -4683.075,E2 -4683.075} C_VEL
LIN {X 0,Y 523.988,Z 318.84,A -85,B 0,C 180,E1 -4686.159,E2 -4686.159} C_VEL
LIN {X 0,Y 523.962,Z 318.834,A -85,B 0,C 180,E1 -4689.262,E2 -4689.262} C_VEL
LIN {X 0,Y 523.983,Z 318.836,A -85,B 0,C 180,E1 -4691.736,E2 -4691.736} C_VEL
LIN {X 0,Y 523.979,Z 318.833,A -85,B 0,C 180,E1 -4695.052,E2 -4695.052} C_VEL
LIN {X 0,Y 523.931,Z 318.847,A -85,B 0,C 180,E1 -4697.97,E2 -4697.97} C_VEL
LIN {X 0,Y 523.944,Z 318.842,A -85,B 0,C 180,E1 -4700.411,E2 -4700.411} C_VEL
LIN {X 0,Y 523.897,Z 318.846,A -85,B 0,C 180,E1 -4702.894,E2 -4702.894} C_VEL
LIN {X 0,Y 523.916,Z 318.844,A -85,B 0,C 180,E1 -4705.42,E2 -4705.42} C_VEL
LIN {X 0,Y 523.905,Z 318.853,A -85,B 0,C 180,E1 -4708.003,E2 -4708.003} C_VEL
LIN {X 0,Y 523.933,Z 318.841,A -85,B 0,C 180,E1 -4710.855,E2 -4710.855} C_VEL
LIN {X 0,Y 523.949,Z 318.846,A -85,B 0,C 180,E1 -4713.735,E2 -4713.735} C_VEL
LIN {X 0,Y 523.909,Z 318.846,A -85,B 0,C 180,E1 -4716.404,E2 -4716.404} C_VEL
LIN {X 0,Y 523.911,Z 318.846,A -85,B 0,C 180,E1 -4719.086,E2 -4719.086} C_VEL
LIN {X 0,Y 523.947,Z 318.843,A -85,B 0,C 180,E1 -4722.119,E2 -4722.119} C_VEL
LIN {X 0,Y 523.947,Z 318.844,A -85,B 0,C 180,E1 -4725.31,E2 -4725.31} C_VEL
LIN {X 0,Y 523.952,Z 318.84,A -85,B 0,C 180,E1 -4728.69,E2 -4728.69} C_VEL
LIN {X 0,Y 523.912,Z 318.849,A -85,B 0,C 180,E1 -4731.081,E2 -4731.081} C_VEL
LIN {X 0,Y 523.922,Z 318.85,A -85,B 0,C 180,E1 -4733.828,E2 -4733.828} C_VEL
LIN {X 0,Y 523.939,Z 318.843,A -85,B 0,C 180,E1 -4736.636,E2 -4736.636} C_VEL
LIN {X 0,Y 523.953,Z 318.848,A -85,B 0,C 180,E1 -4739.356,E2 -4739.356} C_VEL
LIN {X 0,Y 523.974,Z 318.84,A -85,B 0,C 180,E1 -4742.282,E2 -4742.282} C_VEL
LIN {X 0,Y 523.998,Z 318.956,A -85,B 0,C 180,E1 -4744.044,E2 -4744.044} C_VEL
LIN {X 0,Y 525.977,Z 328.337,A -85,B 0,C 180,E1 -4745.531,E2 -4745.531} C_VEL
LIN {X 0,Y 525.754,Z 340.294,A -85,B 0,C 180,E1 -4747.273,E2 -4747.273} C_VEL
LIN {X 0,Y 525.168,Z 361.094,A -85,B 0,C 180,E1 -4750.251,E2 -4750.251} C_VEL
LIN {X 0,Y 524.938,Z 370.847,A -85,B 0,C 180,E1 -4751.631,E2 -4751.631} C_VEL
LIN {X 0,Y 527.17,Z 384.021,A -85,B 0,C 180,E1 -4751.896,E2 -4751.896} C_VEL
LIN {X 0,Y 526.448,Z 509.242,A -85,B 0,C 180,E1 -4753.645,E2 -4753.645} C_VEL
LIN {X 0,Y 526.197,Z 523.473,A -85,B 0,C 180,E1 -4754.001,E2 -4754.001} C_VEL
LIN {X 0,Y 525.924,Z 537.12,A -85,B 0,C 180,E1 -4754.499,E2 -4754.499} C_VEL
LIN {X 0,Y 525.588,Z 549.322,A -85,B 0,C 180,E1 -4755.084,E2 -4755.084} C_VEL
LIN {X 0,Y 525.168,Z 562.162,A -85,B 0,C 180,E1 -4755.864,E2 -4755.864} C_VEL
LIN {X 0,Y 524.813,Z 573.843,A -85,B 0,C 180,E1 -4756.743,E2 -4756.743} C_VEL
LIN {X 0,Y 524.462,Z 584.672,A -85,B 0,C 180,E1 -4757.731,E2 -4757.731} C_VEL
LIN {X 0,Y 524.184,Z 594.341,A -85,B 0,C 180,E1 -4758.79,E2 -4758.79} C_VEL
LIN {X 0,Y 523.88,Z 603.239,A -85,B 0,C 180,E1 -4759.957,E2 -4759.957} C_VEL
LIN {X 0,Y 523.672,Z 611.768,A -85,B 0,C 180,E1 -4761.316,E2 -4761.316} C_VEL
LIN {X 0,Y 523.502,Z 618.642,A -85,B 0,C 180,E1 -4762.673,E2 -4762.673} C_VEL
LIN {X 0,Y 523.473,Z 623.383,A -85,B 0,C 180,E1 -4763.834,E2 -4763.834} C_VEL
LIN {X 0,Y 523.376,Z 627.22,A -85,B 0,C 180,E1 -4764.993,E2 -4764.993} C_VEL
LIN {X 0,Y 523.419,Z 630.18,A -85,B 0,C 180,E1 -4766.151,E2 -4766.151} C_VEL
LIN {X 0,Y 523.333,Z 632.886,A -85,B 0,C 180,E1 -4767.691,E2 -4767.691} C_VEL
LIN {X 0,Y 523.247,Z 634.225,A -85,B 0,C 180,E1 -4769.23,E2 -4769.23} C_VEL
LIN {X 0,Y 523.247,Z 634.226,A -85,B 0,C 180,E1 -4770.77,E2 -4770.77} C_VEL
LIN {X 0,Y 523.333,Z 632.888,A -85,B 0,C 180,E1 -4772.309,E2 -4772.309} C_VEL
LIN {X 0,Y 523.419,Z 630.183,A -85,B 0,C 180,E1 -4773.849,E2 -4773.849} C_VEL
LIN {X 0,Y 523.452,Z 626.032,A -85,B 0,C 180,E1 -4775.393,E2 -4775.393} C_VEL
LIN {X 0,Y 523.494,Z 620.314,A -85,B 0,C 180,E1 -4776.94,E2 -4776.94} C_VEL
LIN {X 0,Y 523.634,Z 613.871,A -85,B 0,C 180,E1 -4778.295,E2 -4778.295} C_VEL
LIN {X 0,Y 523.854,Z 605.867,A -85,B 0,C 180,E1 -4779.654,E2 -4779.654} C_VEL
LIN {X 0,Y 524.106,Z 597.496,A -85,B 0,C 180,E1 -4780.82,E2 -4780.82} C_VEL
LIN {X 0,Y 524.435,Z 586.755,A -85,B 0,C 180,E1 -4782.06,E2 -4782.06} C_VEL
LIN {X 0,Y 524.743,Z 576.185,A -85,B 0,C 180,E1 -4783.062,E2 -4783.062} C_VEL
LIN {X 0,Y 525.136,Z 563.582,A -85,B 0,C 180,E1 -4784.038,E2 -4784.038} C_VEL
LIN {X 0,Y 525.557,Z 551.076,A -85,B 0,C 180,E1 -4784.818,E2 -4784.818} C_VEL
LIN {X 0,Y 525.907,Z 538.224,A -85,B 0,C 180,E1 -4785.452,E2 -4785.452} C_VEL
LIN {X 0,Y 526.17,Z 523.97,A -85,B 0,C 180,E1 -4785.983,E2 -4785.983} C_VEL
LIN {X 0,Y 526.421,Z 510.358,A -85,B 0,C 180,E1 -4786.331,E2 -4786.331} C_VEL
LIN {X 0,Y 526.629,Z 482.234,A -85,B 0,C 180,E1 -4786.748,E2 -4786.748} C_VEL
LIN {X 0,Y 527.15,Z 383.537,A -85,B 0,C 180,E1 -4788.111,E2 -4788.111} C_VEL
LIN {X 0,Y 524.928,Z 370.71,A -85,B 0,C 180,E1 -4788.384,E2 -4788.384} C_VEL
LIN {X 0,Y 525.494,Z 349.675,A -85,B 0,C 180,E1 -4791.373,E2 -4791.373} C_VEL
LIN {X 0,Y 526.06,Z 329.724,A -85,B 0,C 180,E1 -4794.255,E2 -4794.255} C_VEL
LIN {X 0,Y 524.789,Z 322.577,A -85,B 0,C 180,E1 -4795.375,E2 -4795.375} C_VEL
LIN {X 0,Y 523.961,Z 318.846,A -85,B 0,C 180,E1 -4795.979,E2 -4795.979} C_VEL
LIN {X 0,Y 523.937,Z 318.849,A -85,B 0,C 180,E1 -4798.874,E2 -4798.874} C_VEL
LIN {X 0,Y 523.918,Z 318.846,A -85,B 0,C 180,E1 -4801.543,E2 -4801.543} C_VEL
LIN {X 0,Y 523.937,Z 318.849,A -85,B 0,C 180,E1 -4804.289,E2 -4804.289} C_VEL
LIN {X 0,Y 523.907,Z 318.842,A -85,B 0,C 180,E1 -4807.131,E2 -4807.131} C_VEL
LIN {X 0,Y 523.932,Z 318.845,A -85,B 0,C 180,E1 -4810.129,E2 -4810.129} C_VEL
LIN {X 0,Y 523.93,Z 318.847,A -85,B 0,C 180,E1 -4812.458,E2 -4812.458} C_VEL
LIN {X 0,Y 523.947,Z 318.838,A -85,B 0,C 180,E1 -4815.308,E2 -4815.308} C_VEL
